  MoveL 4606 to (37.53, 58.52, -241.21) mm, rotated rx 42.04 ry 15.1 rz -114.75 deg; joints [-18.121, -37.551, 103.007, 143.689, 51.93, -28.848, -355]
  MoveL 4607 to (37.12, 58.35, -241.17) mm, rotated rx 42.04 ry 15.1 rz -114.75 deg; joints [-18.122, -37.581, 103.033, 143.686, 51.926, -28.844, -355]
  MoveL 4608 to (36.72, 58.21, -241.12) mm, rotated rx 42.04 ry 15.1 rz -114.75 deg; joints [-18.121, -37.609, 103.056, 143.684, 51.922, -28.841, -355]
  MoveL 4609 to (36.33, 58.09, -241.05) mm, rotated rx 42.04 ry 15.1 rz -114.75 deg; joints [-18.12, -37.637, 103.078, 143.683, 51.917, -28.837, -355]
  MoveL 4610 to (35.92, 57.93, -241) mm, rotated rx 42.04 ry 15.1 rz -114.75 deg; joints [-18.12, -37.667, 103.103, 143.681, 51.913, -28.833, -355]
  MoveL 4611 to (35.45, 57.73, -240.98) mm, rotated rx 42.04 ry 15.1 rz -114.75 deg; joints [-18.121, -37.701, 103.132, 143.677, 51.91, -28.829, -355]
  MoveL 4612 to (30.23, 55.38, -240.97) mm, rotated rx 42.04 ry 15.1 rz -114.75 deg; joints [-18.146, -38.084, 103.466, 143.625, 51.876, -28.782, -355]
  MoveL 4613 to (29.53, 55.08, -240.96) mm, rotated rx 42.04 ry 15.1 rz -114.75 deg; joints [-18.149, -38.136, 103.51, 143.618, 51.871, -28.775, -355]
  MoveL 4614 to (28.91, 54.84, -240.95) mm, rotated rx 42.04 ry 15.1 rz -114.75 deg; joints [-18.151, -38.179, 103.545, 143.612, 51.865, -28.767, -355]
  MoveL 4615 to (28.35, 54.72, -240.94) mm, rotated rx 42.04 ry 15.1 rz -114.75 deg; joints [-18.152, -38.217, 103.57, 143.604, 51.854, -28.757, -355]
  MoveL 4616 to (27.81, 54.68, -240.9) mm, rotated rx 42.04 ry 15.1 rz -114.75 deg; joints [-18.151, -38.251, 103.587, 143.598, 51.841, -28.745, -355]
  MoveL 4617 to (27.48, 54.71, -240.74) mm, rotated rx 42.04 ry 15.1 rz -114.75 deg; joints [-18.145, -38.271, 103.595, 143.599, 51.83, -28.739, -355]
  MoveL 4618 to (27.48, 54.74, -240.43) mm, rotated rx 42.04 ry 15.1 rz -114.75 deg; joints [-18.133, -38.272, 103.6, 143.614, 51.829, -28.746, -355]
  MoveL 4619 to (27.85, 54.75, -239.94) mm, rotated rx 42.04 ry 15.1 rz -114.75 deg; joints [-18.115, -38.254, 103.6, 143.645, 51.84, -28.768, -355]
  MoveL 4620 to (27.62, 55.34, -238.97) mm, rotated rx 42.04 ry 15.1 rz -114.75 deg; joints [-18.073, -38.258, 103.576, 143.68, 51.806, -28.764, -355]
  MoveL 4621 to (25.78, 55.69, -238.67) mm, rotated rx 42.04 ry 15.1 rz -114.75 deg; joints [-18.06, -38.36, 103.595, 143.657, 51.737, -28.707, -355]
  MoveL 4622 to (23.85, 56.05, -238.46) mm, rotated rx 42.04 ry 15.1 rz -114.75 deg; joints [-18.051, -38.466, 103.614, 143.627, 51.664, -28.646, -355]
  MoveL 4623 to (21.76, 56.41, -238.34) mm, rotated rx 42.04 ry 15.1 rz -114.75 deg; joints [-18.044, -38.581, 103.633, 143.59, 51.586, -28.576, -355]
  MoveL 4624 to (17.55, 57.12, -238.34) mm, rotated rx 42.04 ry 15.1 rz -114.75 deg; joints [-18.041, -38.81, 103.669, 143.503, 51.43, -28.431, -355]
  MoveL 4625 to (15.59, 57.45, -238.25) mm, rotated rx 42.04 ry 15.1 rz -114.75 deg; joints [-18.036, -38.916, 103.687, 143.466, 51.357, -28.366, -355]
  MoveL 4626 to (13.49, 57.8, -238.25) mm, rotated rx 42.04 ry 15.1 rz -114.75 deg; joints [-18.034, -39.031, 103.704, 143.422, 51.279, -28.292, -355]
  MoveL 4627 to (11.38, 58.25, -238.25) mm, rotated rx 42.04 ry 15.1 rz -114.75 deg; joints [-18.032, -39.142, 103.712, 143.376, 51.195, -28.215, -355]
  MoveL 4628 to (8.9, 58.83, -238.07) mm, rotated rx 42.04 ry 15.1 rz -114.75 deg; joints [-18.022, -39.273, 103.721, 143.329, 51.095, -28.126, -355]
  MoveL 4629 to (6.68, 59.07, -237.84) mm, rotated rx 42.04 ry 15.1 rz -114.75 deg; joints [-18.013, -39.398, 103.755, 143.295, 51.019, -28.059, -355]
  MoveL 4630 to (4.53, 59.33, -237.72) mm, rotated rx 42.04 ry 15.1 rz -114.75 deg; joints [-18.007, -39.519, 103.782, 143.257, 50.942, -27.99, -355]
  MoveL 4631 to (2.42, 59.68, -237.61) mm, rotated rx 42.04 ry 15.1 rz -114.75 deg; joints [-18.002, -39.633, 103.799, 143.216, 50.863, -27.918, -355]
  MoveL 4632 to (0.32, 60.02, -237.4) mm, rotated rx 42.04 ry 15.1 rz -114.75 deg; joints [-17.992, -39.748, 103.819, 143.181, 50.785, -27.848, -355]
  MoveL 4633 to (-1.79, 60.37, -237.29) mm, rotated rx 42.04 ry 15.1 rz -114.75 deg; joints [-17.986, -39.863, 103.837, 143.14, 50.705, -27.776, -355]
  MoveL 4634 to (-3.89, 60.71, -237.18) mm, rotated rx 42.04 ry 15.1 rz -114.75 deg; joints [-17.981, -39.977, 103.854, 143.099, 50.626, -27.703, -355]
  MoveL 4635 to (-6, 61.04, -236.97) mm, rotated rx 42.04 ry 15.1 rz -114.75 deg; joints [-17.971, -40.092, 103.874, 143.063, 50.548, -27.633, -355]
  MoveL 4636 to (-8.11, 61.38, -236.86) mm, rotated rx 42.04 ry 15.1 rz -114.75 deg; joints [-17.966, -40.206, 103.891, 143.022, 50.468, -27.56, -355]
  MoveL 4637 to (-10.21, 61.72, -236.76) mm, rotated rx 42.04 ry 15.1 rz -114.75 deg; joints [-17.96, -40.32, 103.907, 142.98, 50.389, -27.486, -355]
  MoveL 4638 to (-12.32, 62.04, -236.55) mm, rotated rx 42.04 ry 15.1 rz -114.75 deg; joints [-17.951, -40.436, 103.928, 142.943, 50.311, -27.416, -355]
  MoveL 4639 to (-14.43, 62.37, -236.45) mm, rotated rx 42.04 ry 15.1 rz -114.75 deg; joints [-17.946, -40.55, 103.944, 142.9, 50.231, -27.342, -355]
  MoveL 4640 to (-16.27, 62.58, -236.19) mm, rotated rx 42.04 ry 15.1 rz -114.75 deg; joints [-17.936, -40.653, 103.968, 142.873, 50.165, -27.284, -355]
  MoveL 4641 to (-17.93, 62.72, -235.82) mm, rotated rx 42.04 ry 15.1 rz -114.75 deg; joints [-17.922, -40.749, 103.997, 142.855, 50.108, -27.238, -355]
  MoveL 4642 to (-19.46, 62.77, -235.32) mm, rotated rx 42.04 ry 15.1 rz -114.75 deg; joints [-17.904, -40.841, 104.034, 142.849, 50.06, -27.203, -355]
  MoveL 4643 to (-18.41, 62.34, -234.48) mm, rotated rx 42.04 ry 15.1 rz -114.75 deg; joints [-17.875, -40.801, 104.069, 142.921, 50.112, -27.276, -355]
  MoveL 4644 to (-18.73, 62.4, -234.45) mm, rotated rx 42.04 ry 15.1 rz -114.75 deg; joints [-17.874, -40.819, 104.071, 142.915, 50.099, -27.264, -355]
  MoveL 4645 to (-19.05, 62.49, -234.41) mm, rotated rx 42.04 ry 15.1 rz -114.75 deg; joints [-17.872, -40.835, 104.071, 142.909, 50.085, -27.252, -355]
  MoveL 4646 to (-19.37, 62.66, -234.35) mm, rotated rx 42.04 ry 15.1 rz -114.75 deg; joints [-17.869, -40.848, 104.063, 142.902, 50.067, -27.237, -355]
  MoveL 4647 to (-19.71, 62.9, -234.31) mm, rotated rx 42.04 ry 15.1 rz -114.75 deg; joints [-17.865, -40.861, 104.05, 142.893, 50.046, -27.218, -355]
  MoveL 4648 to (-20.08, 63.21, -234.29) mm, rotated rx 42.04 ry 15.1 rz -114.75 deg; joints [-17.862, -40.873, 104.03, 142.881, 50.02, -27.195, -355]
  MoveL 4649 to (-23.51, 66.44, -234.29) mm, rotated rx 42.04 ry 15.1 rz -114.75 deg; joints [-17.836, -40.967, 103.812, 142.753, 49.763, -26.96, -355]
  MoveL 4650 to (-23.82, 66.7, -234.26) mm, rotated rx 42.04 ry 15.1 rz -114.75 deg; joints [-17.833, -40.977, 103.796, 142.744, 49.742, -26.941, -355]
  MoveL 4651 to (-24.2, 67.06, -234.26) mm, rotated rx 42.04 ry 15.1 rz -114.75 deg; joints [-17.83, -40.987, 103.771, 142.729, 49.714, -26.915, -355]
  MoveL 4652 to (-24.97, 67.75, -234.22) mm, rotated rx 42.04 ry 15.1 rz -114.75 deg; joints [-17.823, -41.01, 103.726, 142.703, 49.658, -26.865, -355]
  MoveL 4653 to (-26.87, 69.55, -234.22) mm, rotated rx 42.04 ry 15.1 rz -114.75 deg; joints [-17.808, -41.061, 103.604, 142.631, 49.516, -26.733, -355]
  MoveL 4654 to (-27.66, 70.21, -234.21) mm, rotated rx 42.04 ry 15.1 rz -114.75 deg; joints [-17.802, -41.085, 103.56, 142.603, 49.461, -26.682, -355]
  MoveL 4655 to (-28.72, 71.19, -234.27) mm, rotated rx 42.04 ry 15.1 rz -114.75 deg; joints [-17.797, -41.114, 103.493, 142.559, 49.382, -26.608, -355]
  MoveL 4656 to (-29.48, 72.08, -234.53) mm, rotated rx 42.04 ry 15.1 rz -114.75 deg; joints [-17.799, -41.126, 103.422, 142.513, 49.318, -26.541, -355]
  MoveL 4657 to (-29.94, 72.89, -234.97) mm, rotated rx 42.04 ry 15.1 rz -114.75 deg; joints [-17.809, -41.121, 103.35, 142.466, 49.266, -26.481, -355]
  MoveL 4658 to (-30.05, 73.26, -235.26) mm, rotated rx 42.04 ry 15.1 rz -114.75 deg; joints [-17.816, -41.112, 103.312, 142.442, 49.246, -26.455, -355]
  MoveL 4659 to (-30.09, 73.62, -235.59) mm, rotated rx 42.04 ry 15.1 rz -114.75 deg; joints [-17.826, -41.1, 103.275, 142.417, 49.228, -26.43, -355]
  MoveL 4660 to (-29.94, 74.26, -236.4) mm, rotated rx 42.04 ry 15.1 rz -114.75 deg; joints [-17.85, -41.062, 103.197, 142.367, 49.204, -26.386, -355]
  MoveL 4661 to (-29.48, 74.81, -237.4) mm, rotated rx 42.04 ry 15.1 rz -114.75 deg; joints [-17.882, -41.008, 103.117, 142.315, 49.193, -26.349, -355]
  MoveL 4662 to (-27.66, 75.67, -239.96) mm, rotated rx 42.04 ry 15.1 rz -114.75 deg; joints [-17.968, -40.851, 102.951, 142.207, 49.21, -26.3, -355]
  MoveL 4663 to (-25.28, 75.96, -242.53) mm, rotated rx 42.04 ry 15.1 rz -114.75 deg; joints [-18.059, -40.68, 102.822, 142.12, 49.269, -26.29, -355]
  MoveL 4664 to (-23, 75.48, -244.36) mm, rotated rx 42.04 ry 15.1 rz -114.75 deg; joints [-18.129, -40.547, 102.78, 142.084, 49.361, -26.329, -355]
  MoveL 4665 to (-21.89, 74.94, -245) mm, rotated rx 42.04 ry 15.1 rz -114.75 deg; joints [-18.157, -40.495, 102.792, 142.084, 49.42, -26.368, -355]
  MoveL 4666 to (-20.81, 74.21, -245.46) mm, rotated rx 42.04 ry 15.1 rz -114.75 deg; joints [-18.18, -40.453, 102.826, 142.097, 49.486, -26.418, -355]
  MoveL 4667 to (-18.73, 72.17, -245.82) mm, rotated rx 42.04 ry 15.1 rz -114.75 deg; joints [-18.21, -40.396, 102.958, 142.159, 49.644, -26.556, -355]
  MoveL 4668 to (-16.71, 69.76, -245.82) mm, rotated rx 42.04 ry 15.1 rz -114.75 deg; joints [-18.23, -40.358, 103.132, 142.245, 49.817, -26.717, -355]
  MoveL 4669 to (-16.04, 68.99, -245.84) mm, rotated rx 42.04 ry 15.1 rz -114.75 deg; joints [-18.237, -40.344, 103.186, 142.272, 49.873, -26.768, -355]
  MoveL 4670 to (-15.37, 68.19, -245.84) mm, rotated rx 42.04 ry 15.1 rz -114.75 deg; joints [-18.244, -40.331, 103.244, 142.3, 49.93, -26.821, -355]
  MoveL 4671 to (-15.04, 67.81, -245.84) mm, rotated rx 42.04 ry 15.1 rz -114.75 deg; joints [-18.247, -40.325, 103.271, 142.313, 49.958, -26.846, -355]
  MoveL 4672 to (-14.61, 67.31, -245.87) mm, rotated rx 42.04 ry 15.1 rz -114.75 deg; joints [-18.253, -40.316, 103.306, 142.33, 49.994, -26.879, -355]
  MoveL 4673 to (-14.2, 66.87, -245.93) mm, rotated rx 42.04 ry 15.1 rz -114.75 deg; joints [-18.258, -40.306, 103.335, 142.343, 50.027, -26.908, -355]
  MoveL 4674 to (-13.85, 66.51, -246) mm, rotated rx 42.04 ry 15.1 rz -114.75 deg; joints [-18.264, -40.296, 103.358, 142.353, 50.054, -26.931, -355]
  MoveL 4675 to (-13.52, 66.18, -246.05) mm, rotated rx 42.04 ry 15.1 rz -114.75 deg; joints [-18.269, -40.287, 103.38, 142.363, 50.08, -26.953, -355]
  MoveL 4676 to (-13.21, 65.84, -246.08) mm, rotated rx 42.04 ry 15.1 rz -114.75 deg; joints [-18.273, -40.28, 103.403, 142.373, 50.105, -26.975, -355]
  MoveL 4677 to (-12.2, 64.63, -246.08) mm, rotated rx 42.04 ry 15.1 rz -114.75 deg; joints [-18.283, -40.26, 103.489, 142.415, 50.192, -27.055, -355]
  MoveL 4678 to (-11.86, 64.26, -246.1) mm, rotated rx 42.04 ry 15.1 rz -114.75 deg; joints [-18.287, -40.252, 103.514, 142.428, 50.219, -27.08, -355]
  MoveL 4679 to (-11.55, 63.95, -246.13) mm, rotated rx 42.04 ry 15.1 rz -114.75 deg; joints [-18.29, -40.244, 103.535, 142.438, 50.243, -27.101, -355]
  MoveL 4680 to (-11.26, 63.7, -246.17) mm, rotated rx 42.04 ry 15.1 rz -114.75 deg; joints [-18.294, -40.234, 103.55, 142.446, 50.264, -27.118, -355]
  MoveL 4681 to (-10.99, 63.56, -246.24) mm, rotated rx 42.04 ry 15.1 rz -114.75 deg; joints [-18.298, -40.222, 103.555, 142.451, 50.278, -27.13, -355]
  MoveL 4682 to (-10.73, 63.46, -246.31) mm, rotated rx 42.04 ry 15.1 rz -114.75 deg; joints [-18.301, -40.21, 103.557, 142.454, 50.29, -27.14, -355]
  MoveL 4683 to (-11.92, 64.52, -247.11) mm, rotated rx 42.04 ry 15.1 rz -114.75 deg; joints [-18.322, -40.238, 103.47, 142.371, 50.205, -27.039, -355]
  MoveL 4684 to (-10.23, 63.99, -247.52) mm, rotated rx 42.04 ry 15.1 rz -114.75 deg; joints [-18.341, -40.153, 103.473, 142.393, 50.28, -27.101, -355]
  MoveL 4685 to (-8.44, 63.45, -247.78) mm, rotated rx 42.04 ry 15.1 rz -114.75 deg; joints [-18.354, -40.062, 103.477, 142.425, 50.359, -27.17, -355]
  MoveL 4686 to (-6.51, 62.9, -247.96) mm, rotated rx 42.04 ry 15.1 rz -114.75 deg; joints [-18.364, -39.965, 103.481, 142.464, 50.442, -27.245, -355]
  MoveL 4687 to (-4.46, 62.34, -248.16) mm, rotated rx 42.04 ry 15.1 rz -114.75 deg; joints [-18.375, -39.861, 103.483, 142.504, 50.529, -27.324, -355]
  MoveL 4688 to (-2.4, 61.76, -248.25) mm, rotated rx 42.04 ry 15.1 rz -114.75 deg; joints [-18.383, -39.758, 103.489, 142.55, 50.617, -27.406, -355]
  MoveL 4689 to (-0.35, 61.17, -248.35) mm, rotated rx 42.04 ry 15.1 rz -114.75 deg; joints [-18.39, -39.655, 103.494, 142.595, 50.705, -27.488, -355]
  MoveL 4690 to (1.71, 60.6, -248.55) mm, rotated rx 42.04 ry 15.1 rz -114.75 deg; joints [-18.401, -39.55, 103.496, 142.635, 50.793, -27.566, -355]
  MoveL 4691 to (3.76, 60.01, -248.65) mm, rotated rx 42.04 ry 15.1 rz -114.75 deg; joints [-18.409, -39.447, 103.501, 142.679, 50.881, -27.647, -355]
  MoveL 4692 to (5.81, 59.42, -248.75) mm, rotated rx 42.04 ry 15.1 rz -114.75 deg; joints [-18.416, -39.343, 103.505, 142.723, 50.969, -27.728, -355]
  MoveL 4693 to (7.86, 58.83, -248.95) mm, rotated rx 42.04 ry 15.1 rz -114.75 deg; joints [-18.428, -39.239, 103.507, 142.762, 51.056, -27.806, -355]
  MoveL 4694 to (11.96, 57.64, -249.15) mm, rotated rx 42.04 ry 15.1 rz -114.75 deg; joints [-18.443, -39.032, 103.515, 142.849, 51.232, -27.966, -355]
  MoveL 4695 to (13.68, 57.13, -249.36) mm, rotated rx 42.04 ry 15.1 rz -114.75 deg; joints [-18.454, -38.944, 103.516, 142.879, 51.306, -28.03, -355]
  MoveL 4696 to (15.57, 56.62, -249.43) mm, rotated rx 42.04 ry 15.1 rz -114.75 deg; joints [-18.46, -38.846, 103.516, 142.919, 51.385, -28.103, -355]
  MoveL 4697 to (17.57, 56.14, -249.44) mm, rotated rx 42.04 ry 15.1 rz -114.75 deg; joints [-18.464, -38.742, 103.512, 142.963, 51.466, -28.178, -355]
  MoveL 4698 to (20.13, 55.38, -249.55) mm, rotated rx 42.04 ry 15.1 rz -114.75 deg; joints [-18.473, -38.612, 103.517, 143.016, 51.576, -28.278, -355]
  MoveL 4699 to (22.57, 54.54, -249.64) mm, rotated rx 42.04 ry 15.1 rz -114.75 deg; joints [-18.482, -38.492, 103.532, 143.07, 51.686, -28.378, -355]
  MoveL 4700 to (24.68, 53.87, -249.74) mm, rotated rx 42.04 ry 15.1 rz -114.75 deg; joints [-18.49, -38.386, 103.538, 143.113, 51.778, -28.46, -355]
  MoveL 4701 to (26.64, 53.28, -249.91) mm, rotated rx 42.04 ry 15.1 rz -114.75 deg; joints [-18.501, -38.286, 103.54, 143.149, 51.862, -28.534, -355]
  MoveL 4702 to (28.45, 52.71, -250.19) mm, rotated rx 42.04 ry 15.1 rz -114.75 deg; joints [-18.515, -38.192, 103.54, 143.177, 51.941, -28.599, -355]
  MoveL 4703 to (30.26, 52.15, -250.48) mm, rotated rx 42.04 ry 15.1 rz -114.75 deg; joints [-18.53, -38.099, 103.54, 143.203, 52.019, -28.664, -355]
  MoveL 4704 to (32.04, 51.55, -250.77) mm, rotated rx 42.04 ry 15.1 rz -114.75 deg; joints [-18.545, -38.007, 103.543, 143.229, 52.098, -28.729, -355]
  MoveL 4705 to (33.94, 50.95, -250.93) mm, rotated rx 42.04 ry 15.1 rz -114.75 deg; joints [-18.555, -37.91, 103.545, 143.264, 52.18, -28.8, -355]
  MoveL 4706 to (34.26, 50.38, -251.55) mm, rotated rx 42.04 ry 15.1 rz -114.75 deg; joints [-18.583, -37.903, 103.573, 143.248, 52.216, -28.815, -355]
  MoveL 4707 to (33.95, 50.33, -251.86) mm, rotated rx 42.04 ry 15.1 rz -114.75 deg; joints [-18.595, -37.92, 103.579, 143.228, 52.209, -28.801, -355]
  MoveL 4708 to (33.93, 50.29, -252.05) mm, rotated rx 42.04 ry 15.1 rz -114.75 deg; joints [-18.603, -37.921, 103.579, 143.218, 52.21, -28.797, -355]
  MoveL 4709 to (34.18, 50.27, -252.15) mm, rotated rx 42.04 ry 15.1 rz -114.75 deg; joints [-18.607, -37.906, 103.572, 143.218, 52.218, -28.802, -355]
  MoveL 4710 to (34.62, 50.32, -252.17) mm, rotated rx 42.04 ry 15.1 rz -114.75 deg; joints [-18.606, -37.878, 103.556, 143.224, 52.228, -28.812, -355]
  MoveL 4711 to (35.1, 50.41, -252.17) mm, rotated rx 42.04 ry 15.1 rz -114.75 deg; joints [-18.605, -37.846, 103.536, 143.231, 52.237, -28.821, -355]
  MoveL 4712 to (36.04, 50.7, -252.2) mm, rotated rx 42.04 ry 15.1 rz -114.75 deg; joints [-18.603, -37.781, 103.487, 143.241, 52.249, -28.834, -355]
  MoveL 4713 to (37.53, 51.18, -252.2) mm, rotated rx 42.04 ry 15.1 rz -114.75 deg; joints [-18.598, -37.677, 103.409, 143.259, 52.269, -28.855, -355]
  MoveL 4714 to (38.48, 51.44, -252.22) mm, rotated rx 42.04 ry 15.1 rz -114.75 deg; joints [-18.595, -37.613, 103.362, 143.27, 52.282, -28.87, -355]
  MoveL 4715 to (39.48, 51.75, -252.22) mm, rotated rx 42.04 ry 15.1 rz -114.75 deg; joints [-18.591, -37.543, 103.31, 143.283, 52.295, -28.884, -355]
  MoveL 4716 to (39.97, 51.9, -252.23) mm, rotated rx 42.04 ry 15.1 rz -114.75 deg; joints [-18.59, -37.509, 103.284, 143.288, 52.301, -28.891, -355]
  MoveL 4717 to (40.42, 52.03, -252.26) mm, rotated rx 42.04 ry 15.1 rz -114.75 deg; joints [-18.59, -37.478, 103.261, 143.292, 52.308, -28.897, -355]
  MoveL 4718 to (40.85, 52.14, -252.31) mm, rotated rx 42.04 ry 15.1 rz -114.75 deg; joints [-18.59, -37.449, 103.24, 143.295, 52.314, -28.903, -355]
  MoveL 4719 to (41.24, 52.24, -252.37) mm, rotated rx 42.04 ry 15.1 rz -114.75 deg; joints [-18.591, -37.422, 103.22, 143.297, 52.32, -28.908, -355]
  MoveL 4720 to (41.65, 52.34, -252.43) mm, rotated rx 42.04 ry 15.1 rz -114.75 deg; joints [-18.592, -37.394, 103.2, 143.3, 52.327, -28.914, -355]
  MoveL 4721 to (42.09, 52.46, -252.46) mm, rotated rx 42.04 ry 15.1 rz -114.75 deg; joints [-18.592, -37.363, 103.177, 143.304, 52.333, -28.92, -355]
  MoveL 4722 to (42.55, 52.59, -252.48) mm, rotated rx 42.04 ry 15.1 rz -114.75 deg; joints [-18.591, -37.331, 103.154, 143.308, 52.339, -28.926, -355]
  MoveL 4723 to (42.98, 52.7, -252.53) mm, rotated rx 42.04 ry 15.1 rz -114.75 deg; joints [-18.591, -37.303, 103.133, 143.312, 52.346, -28.932, -355]
  MoveL 4724 to (43.37, 52.78, -252.59) mm, rotated rx 42.04 ry 15.1 rz -114.75 deg; joints [-18.593, -37.276, 103.115, 143.314, 52.353, -28.938, -355]
  MoveL 4725 to (43.77, 52.87, -252.64) mm, rotated rx 42.04 ry 15.1 rz -114.75 deg; joints [-18.593, -37.249, 103.095, 143.317, 52.359, -28.944, -355]
  MoveL 4726 to (44.2, 52.98, -252.67) mm, rotated rx 42.04 ry 15.1 rz -114.75 deg; joints [-18.593, -37.22, 103.074, 143.321, 52.366, -28.95, -355]
  MoveL 4727 to (44.7, 53.14, -252.67) mm, rotated rx 42.04 ry 15.1 rz -114.75 deg; joints [-18.591, -37.185, 103.048, 143.327, 52.372, -28.957, -355]
  MoveL 4728 to (47.54, 53.78, -253.03) mm, rotated rx 42.04 ry 15.1 rz -114.75 deg; joints [-18.597, -36.992, 102.912, 143.347, 52.419, -28.997, -355]
  MoveL 4729 to (48.83, 53.85, -253.47) mm, rotated rx 42.04 ry 15.1 rz -114.75 deg; joints [-18.611, -36.909, 102.862, 143.345, 52.449, -29.017, -355]
  MoveL 4730 to (50.03, 53.76, -254.09) mm, rotated rx 42.04 ry 15.1 rz -114.75 deg; joints [-18.634, -36.834, 102.825, 143.335, 52.485, -29.036, -355]
  MoveL 4731 to (52.15, 53.11, -255.87) mm, rotated rx 42.04 ry 15.1 rz -114.75 deg; joints [-18.705, -36.711, 102.788, 143.293, 52.571, -29.071, -355]
  MoveL 4732 to (53.9, 51.8, -258.37) mm, rotated rx 42.04 ry 15.1 rz -114.75 deg; joints [-18.809, -36.622, 102.8, 143.219, 52.677, -29.105, -355]
  MoveL 4733 to (54.89, 50.3, -260.86) mm, rotated rx 42.04 ry 15.1 rz -114.75 deg; joints [-18.915, -36.585, 102.849, 143.135, 52.772, -29.127, -355]
  MoveL 4734 to (54.95, 49.65, -261.84) mm, rotated rx 42.04 ry 15.1 rz -114.75 deg; joints [-18.957, -36.592, 102.882, 143.097, 52.803, -29.13, -355]
  MoveL 4735 to (54.71, 49.05, -262.64) mm, rotated rx 42.04 ry 15.1 rz -114.75 deg; joints [-18.993, -36.617, 102.922, 143.063, 52.823, -29.126, -355]
  MoveL 4736 to (54.48, 48.78, -262.98) mm, rotated rx 42.04 ry 15.1 rz -114.75 deg; joints [-19.008, -36.635, 102.944, 143.047, 52.83, -29.123, -355]
  MoveL 4737 to (54.18, 48.53, -263.27) mm, rotated rx 42.04 ry 15.1 rz -114.75 deg; joints [-19.021, -36.659, 102.967, 143.032, 52.833, -29.118, -355]
  MoveL 4738 to (53.36, 48.06, -263.71) mm, rotated rx 42.04 ry 15.1 rz -114.75 deg; joints [-19.043, -36.718, 103.019, 143.003, 52.832, -29.103, -355]
  MoveL 4739 to (52.24, 47.66, -263.98) mm, rotated rx 42.04 ry 15.1 rz -114.75 deg; joints [-19.058, -36.795, 103.077, 142.977, 52.821, -29.083, -355]
  MoveL 4740 to (50.83, 47.32, -264.07) mm, rotated rx 42.04 ry 15.1 rz -114.75 deg; joints [-19.065, -36.889, 103.14, 142.955, 52.799, -29.057, -355]
  MoveL 4741 to (48.26, 46.82, -264.07) mm, rotated rx 42.04 ry 15.1 rz -114.75 deg; joints [-19.072, -37.058, 103.25, 142.919, 52.753, -29.009, -355]
  MoveL 4742 to (47.82, 46.75, -264.04) mm, rotated rx 42.04 ry 15.1 rz -114.75 deg; joints [-19.072, -37.086, 103.268, 142.915, 52.744, -29.001, -355]
  MoveL 4743 to (47.42, 46.7, -263.99) mm, rotated rx 42.04 ry 15.1 rz -114.75 deg; joints [-19.071, -37.113, 103.284, 142.911, 52.736, -28.994, -355]
  MoveL 4744 to (47.04, 46.66, -263.92) mm, rotated rx 42.04 ry 15.1 rz -114.75 deg; joints [-19.069, -37.138, 103.299, 142.909, 52.727, -28.987, -355]
  MoveL 4745 to (46.61, 46.6, -263.87) mm, rotated rx 42.04 ry 15.1 rz -114.75 deg; joints [-19.068, -37.165, 103.316, 142.905, 52.719, -28.979, -355]
  MoveL 4746 to (46.12, 46.52, -263.83) mm, rotated rx 42.04 ry 15.1 rz -114.75 deg; joints [-19.068, -37.198, 103.336, 142.9, 52.709, -28.97, -355]
  MoveL 4747 to (45.6, 46.45, -263.77) mm, rotated rx 42.04 ry 15.1 rz -114.75 deg; joints [-19.067, -37.231, 103.357, 142.895, 52.698, -28.961, -355]
  MoveL 4748 to (45.06, 46.36, -263.76) mm, rotated rx 42.04 ry 15.1 rz -114.75 deg; joints [-19.067, -37.266, 103.379, 142.888, 52.688, -28.951, -355]
  MoveL 4749 to (44.43, 46.23, -263.77) mm, rotated rx 42.04 ry 15.1 rz -114.75 deg; joints [-19.07, -37.308, 103.406, 142.879, 52.677, -28.938, -355]
  MoveL 4750 to (43.59, 46.04, -263.84) mm, rotated rx 42.04 ry 15.1 rz -114.75 deg; joints [-19.075, -37.364, 103.442, 142.864, 52.663, -28.922, -355]
  MoveL 4751 to (43.07, 45.94, -263.84) mm, rotated rx 42.04 ry 15.1 rz -114.75 deg; joints [-19.076, -37.398, 103.464, 142.857, 52.653, -28.912, -355]
  MoveL 4752 to (42.58, 45.85, -263.83) mm, rotated rx 42.04 ry 15.1 rz -114.75 deg; joints [-19.077, -37.43, 103.484, 142.85, 52.644, -28.903, -355]
  MoveL 4753 to (42.12, 45.77, -263.81) mm, rotated rx 42.04 ry 15.1 rz -114.75 deg; joints [-19.077, -37.46, 103.503, 142.845, 52.635, -28.894, -355]
  MoveL 4754 to (41.71, 45.71, -263.76) mm, rotated rx 42.04 ry 15.1 rz -114.75 deg; joints [-19.076, -37.487, 103.52, 142.841, 52.626, -28.886, -355]
  MoveL 4755 to (41.31, 45.68, -263.7) mm, rotated rx 42.04 ry 15.1 rz -114.75 deg; joints [-19.075, -37.512, 103.534, 142.838, 52.617, -28.878, -355]
  MoveL 4756 to (40.89, 45.69, -263.65) mm, rotated rx 42.04 ry 15.1 rz -114.75 deg; joints [-19.073, -37.538, 103.545, 142.833, 52.605, -28.868, -355]
  MoveL 4757 to (40.48, 45.74, -263.59) mm, rotated rx 42.04 ry 15.1 rz -114.75 deg; joints [-19.071, -37.561, 103.552, 142.828, 52.591, -28.856, -355]
  MoveL 4758 to (40.27, 45.83, -263.43) mm, rotated rx 42.04 ry 15.1 rz -114.75 deg; joints [-19.064, -37.573, 103.553, 142.831, 52.582, -28.851, -355]
  MoveL 4759 to (40.37, 45.89, -263.12) mm, rotated rx 42.04 ry 15.1 rz -114.75 deg; joints [-19.052, -37.568, 103.553, 142.847, 52.582, -28.86, -355]
  MoveL 4760 to (40.81, 45.91, -262.62) mm, rotated rx 42.04 ry 15.1 rz -114.75 deg; joints [-19.033, -37.546, 103.552, 142.879, 52.595, -28.884, -355]
  MoveL 4761 to (39.98, 46.22, -261.77) mm, rotated rx 42.04 ry 15.1 rz -114.75 deg; joints [-18.999, -37.594, 103.565, 142.902, 52.558, -28.871, -355]
  MoveL 4762 to (36.04, 47.87, -261.77) mm, rotated rx 42.04 ry 15.1 rz -114.75 deg; joints [-18.986, -37.781, 103.518, 142.809, 52.369, -28.698, -355]
  MoveL 4763 to (34.2, 48.65, -261.71) mm, rotated rx 42.04 ry 15.1 rz -114.75 deg; joints [-18.978, -37.869, 103.497, 142.768, 52.28, -28.618, -355]
  MoveL 4764 to (32.37, 49.43, -261.56) mm, rotated rx 42.04 ry 15.1 rz -114.75 deg; joints [-18.966, -37.956, 103.476, 142.73, 52.191, -28.54, -355]
  MoveL 4765 to (30.26, 50.34, -261.36) mm, rotated rx 42.04 ry 15.1 rz -114.75 deg; joints [-18.952, -38.057, 103.452, 142.689, 52.088, -28.451, -355]
  MoveL 4766 to (28.27, 51.2, -261.15) mm, rotated rx 42.04 ry 15.1 rz -114.75 deg; joints [-18.937, -38.152, 103.43, 142.65, 51.991, -28.367, -355]
  MoveL 4767 to (26.26, 52.05, -261.05) mm, rotated rx 42.04 ry 15.1 rz -114.75 deg; joints [-18.927, -38.247, 103.406, 142.605, 51.894, -28.279, -355]
  MoveL 4768 to (24.29, 52.87, -261.05) mm, rotated rx 42.04 ry 15.1 rz -114.75 deg; joints [-18.921, -38.339, 103.38, 142.557, 51.799, -28.191, -355]
  MoveL 4769 to (22.46, 53.64, -260.98) mm, rotated rx 42.04 ry 15.1 rz -114.75 deg; joints [-18.912, -38.425, 103.358, 142.514, 51.71, -28.11, -355]
  MoveL 4770 to (20.73, 54.36, -260.86) mm, rotated rx 42.04 ry 15.1 rz -114.75 deg; joints [-18.903, -38.507, 103.338, 142.477, 51.627, -28.035, -355]
  MoveL 4771 to (18.84, 55.15, -260.8) mm, rotated rx 42.04 ry 15.1 rz -114.75 deg; joints [-18.894, -38.596, 103.314, 142.432, 51.536, -27.952, -355]
  MoveL 4772 to (16.87, 55.97, -260.62) mm, rotated rx 42.04 ry 15.1 rz -114.75 deg; joints [-18.881, -38.689, 103.291, 142.391, 51.441, -27.867, -355]
  MoveL 4773 to (12.93, 57.61, -260.44) mm, rotated rx 42.04 ry 15.1 rz -114.75 deg; joints [-18.862, -38.873, 103.241, 142.299, 51.25, -27.692, -355]
  MoveL 4774 to (10.96, 58.43, -260.26) mm, rotated rx 42.04 ry 15.1 rz -114.75 deg; joints [-18.849, -38.966, 103.218, 142.258, 51.155, -27.607, -355]
  MoveL 4775 to (8.98, 59.24, -260.08) mm, rotated rx 42.04 ry 15.1 rz -114.75 deg; joints [-18.836, -39.059, 103.195, 142.215, 51.06, -27.521, -355]
  MoveL 4776 to (7.02, 60.06, -260.08) mm, rotated rx 42.04 ry 15.1 rz -114.75 deg; joints [-18.83, -39.149, 103.166, 142.164, 50.964, -27.43, -355]
  MoveL 4777 to (5.04, 60.87, -259.9) mm, rotated rx 42.04 ry 15.1 rz -114.75 deg; joints [-18.817, -39.242, 103.143, 142.121, 50.869, -27.344, -355]
  MoveL 4778 to (3.06, 61.67, -259.72) mm, rotated rx 42.04 ry 15.1 rz -114.75 deg; joints [-18.805, -39.334, 103.12, 142.077, 50.774, -27.258, -355]
  MoveL 4779 to (1.09, 62.49, -259.72) mm, rotated rx 42.04 ry 15.1 rz -114.75 deg; joints [-18.799, -39.424, 103.09, 142.025, 50.679, -27.166, -355]
  MoveL 4780 to (-0.73, 63.18, -259.53) mm, rotated rx 42.04 ry 15.1 rz -114.75 deg; joints [-18.786, -39.511, 103.073, 141.987, 50.594, -27.089, -355]
  MoveL 4781 to (-2.36, 63.72, -259.21) mm, rotated rx 42.04 ry 15.1 rz -114.75 deg; joints [-18.771, -39.592, 103.068, 141.962, 50.521, -27.027, -355]
  MoveL 4782 to (-3.83, 64.12, -258.74) mm, rotated rx 42.04 ry 15.1 rz -114.75 deg; joints [-18.751, -39.67, 103.074, 141.949, 50.459, -26.979, -355]
  MoveL 4783 to (-3.04, 63.61, -257.98) mm, rotated rx 42.04 ry 15.1 rz -114.75 deg; joints [-18.727, -39.647, 103.121, 142.013, 50.507, -27.045, -355]
  MoveL 4784 to (-3.4, 63.81, -257.97) mm, rotated rx 42.04 ry 15.1 rz -114.75 deg; joints [-18.725, -39.662, 103.111, 142.002, 50.487, -27.026, -355]
  MoveC 4785 to (-5.59, 66.61, -257.97) mm, rotated rx 42.04 ry 15.1 rz -114.75 deg; joints [-18.701, -39.7, 102.909, 141.909, 50.292, -26.846, -355] to (-7.54, 69.58, -257.97) mm, rotated rx 42.04 ry 15.1 rz -114.75 deg; joints [-18.674, -39.717, 102.687, 141.817, 50.096, -26.665, -355]
  MoveL 4786 to (-7.54, 69.58, -257.97) mm, rotated rx 42.04 ry 15.1 rz -114.75 deg; joints [-18.674, -39.717, 102.687, 141.817, 50.096, -26.665, -355]
  MoveL 4787 to (-7.81, 69.96, -257.95) mm, rotated rx 42.04 ry 15.1 rz -114.75 deg; joints [-18.67, -39.721, 102.658, 141.805, 50.07, -26.642, -355]
  MoveL 4788 to (-8.07, 70.3, -257.9) mm, rotated rx 42.04 ry 15.1 rz -114.75 deg; joints [-18.665, -39.725, 102.635, 141.797, 50.047, -26.622, -355]
  MoveL 4789 to (-8.32, 70.62, -257.84) mm, rotated rx 42.04 ry 15.1 rz -114.75 deg; joints [-18.66, -39.73, 102.613, 141.789, 50.024, -26.602, -355]
  MoveL 4790 to (-8.58, 70.97, -257.79) mm, rotated rx 42.04 ry 15.1 rz -114.75 deg; joints [-18.656, -39.734, 102.589, 141.779, 50, -26.581, -355]
  MoveL 4791 to (-8.85, 71.35, -257.76) mm, rotated rx 42.04 ry 15.1 rz -114.75 deg; joints [-18.651, -39.738, 102.561, 141.768, 49.974, -26.558, -355]
  MoveL 4792 to (-9.15, 71.78, -257.75) mm, rotated rx 42.04 ry 15.1 rz -114.75 deg; joints [-18.647, -39.741, 102.529, 141.755, 49.946, -26.532, -355]
  MoveL 4793 to (-9.72, 72.66, -257.75) mm, rotated rx 42.04 ry 15.1 rz -114.75 deg; joints [-18.639, -39.746, 102.463, 141.728, 49.888, -26.478, -355]
  MoveL 4794 to (-10.48, 73.9, -257.84) mm, rotated rx 42.04 ry 15.1 rz -114.75 deg; joints [-18.632, -39.748, 102.366, 141.685, 49.808, -26.401, -355]
  MoveL 4795 to (-10.99, 74.99, -258.11) mm, rotated rx 42.04 ry 15.1 rz -114.75 deg; joints [-18.632, -39.739, 102.273, 141.64, 49.742, -26.332, -355]
  MoveL 4796 to (-11.26, 75.92, -258.57) mm, rotated rx 42.04 ry 15.1 rz -114.75 deg; joints [-18.641, -39.72, 102.185, 141.594, 49.691, -26.273, -355]
  MoveL 4797 to (-11.28, 76.69, -259.21) mm, rotated rx 42.04 ry 15.1 rz -114.75 deg; joints [-18.657, -39.69, 102.102, 141.546, 49.654, -26.222, -355]
  MoveL 4798 to (-11.07, 77.3, -260.03) mm, rotated rx 42.04 ry 15.1 rz -114.75 deg; joints [-18.681, -39.649, 102.024, 141.497, 49.632, -26.179, -355]
  MoveL 4799 to (-10.62, 77.75, -261.04) mm, rotated rx 42.04 ry 15.1 rz -114.75 deg; joints [-18.714, -39.598, 101.951, 141.447, 49.624, -26.146, -355]
  MoveL 4800 to (-8.98, 78.18, -263.6) mm, rotated rx 42.04 ry 15.1 rz -114.75 deg; joints [-18.803, -39.465, 101.82, 141.342, 49.651, -26.105, -355]
  MoveL 4801 to (-6.94, 77.93, -266.16) mm, rotated rx 42.04 ry 15.1 rz -114.75 deg; joints [-18.897, -39.331, 101.74, 141.258, 49.721, -26.105, -355]
  MoveL 4802 to (-5.99, 77.53, -267.16) mm, rotated rx 42.04 ry 15.1 rz -114.75 deg; joints [-18.937, -39.279, 101.733, 141.234, 49.767, -26.123, -355]
  MoveL 4803 to (-5.08, 76.94, -267.99) mm, rotated rx 42.04 ry 15.1 rz -114.75 deg; joints [-18.972, -39.237, 101.746, 141.222, 49.82, -26.152, -355]
  MoveL 4804 to (-4.2, 76.17, -268.63) mm, rotated rx 42.04 ry 15.1 rz -114.75 deg; joints [-19.002, -39.206, 101.782, 141.221, 49.881, -26.192, -355]
  MoveL 4805 to (-3.37, 75.22, -269.08) mm, rotated rx 42.04 ry 15.1 rz -114.75 deg; joints [-19.027, -39.184, 101.839, 141.233, 49.949, -26.245, -355]
  MoveL 4806 to (-1.84, 72.76, -269.45) mm, rotated rx 42.04 ry 15.1 rz -114.75 deg; joints [-19.062, -39.172, 102.016, 141.29, 50.108, -26.383, -355]
  MoveL 4807 to (-1.36, 71.83, -269.45) mm, rotated rx 42.04 ry 15.1 rz -114.75 deg; joints [-19.071, -39.174, 102.089, 141.317, 50.165, -26.437, -355]
  MoveL 4808 to (-1.12, 71.36, -269.46) mm, rotated rx 42.04 ry 15.1 rz -114.75 deg; joints [-19.075, -39.175, 102.125, 141.33, 50.194, -26.463, -355]
  MoveL 4809 to (-0.89, 70.95, -269.48) mm, rotated rx 42.04 ry 15.1 rz -114.75 deg; joints [-19.08, -39.175, 102.157, 141.341, 50.22, -26.487, -355]
  MoveL 4810 to (-0.67, 70.58, -269.53) mm, rotated rx 42.04 ry 15.1 rz -114.75 deg; joints [-19.085, -39.174, 102.183, 141.35, 50.243, -26.507, -355]
  MoveL 4811 to (-0.46, 70.24, -269.58) mm, rotated rx 42.04 ry 15.1 rz -114.75 deg; joints [-19.09, -39.172, 102.208, 141.357, 50.265, -26.526, -355]
  MoveL 4812 to (-0.24, 69.88, -269.63) mm, rotated rx 42.04 ry 15.1 rz -114.75 deg; joints [-19.095, -39.171, 102.234, 141.366, 50.288, -26.546, -355]
  MoveL 4813 to (-0.02, 69.47, -269.65) mm, rotated rx 42.04 ry 15.1 rz -114.75 deg; joints [-19.1, -39.171, 102.265, 141.376, 50.314, -26.57, -355]
  MoveL 4814 to (0.21, 69.03, -269.66) mm, rotated rx 42.04 ry 15.1 rz -114.75 deg; joints [-19.104, -39.172, 102.3, 141.389, 50.341, -26.595, -355]
  MoveL 4815 to (0.46, 68.53, -269.65) mm, rotated rx 42.04 ry 15.1 rz -114.75 deg; joints [-19.108, -39.173, 102.338, 141.403, 50.371, -26.623, -355]
  MoveL 4816 to (0.71, 68.06, -269.66) mm, rotated rx 42.04 ry 15.1 rz -114.75 deg; joints [-19.113, -39.174, 102.374, 141.416, 50.4, -26.65, -355]
  MoveL 4817 to (0.94, 67.63, -269.68) mm, rotated rx 42.04 ry 15.1 rz -114.75 deg; joints [-19.118, -39.174, 102.407, 141.427, 50.427, -26.674, -355]
  MoveL 4818 to (1.18, 67.22, -269.73) mm, rotated rx 42.04 ry 15.1 rz -114.75 deg; joints [-19.123, -39.173, 102.438, 141.437, 50.453, -26.697, -355]
  MoveL 4819 to (1.44, 66.79, -269.81) mm, rotated rx 42.04 ry 15.1 rz -114.75 deg; joints [-19.13, -39.171, 102.468, 141.446, 50.481, -26.72, -355]
  MoveL 4820 to (1.75, 66.27, -269.87) mm, rotated rx 42.04 ry 15.1 rz -114.75 deg; joints [-19.137, -39.168, 102.506, 141.458, 50.514, -26.749, -355]
  MoveL 4821 to (2.02, 65.77, -269.89) mm, rotated rx 42.04 ry 15.1 rz -114.75 deg; joints [-19.142, -39.168, 102.544, 141.471, 50.546, -26.778, -355]
  MoveL 4822 to (2.27, 65.3, -269.89) mm, rotated rx 42.04 ry 15.1 rz -114.75 deg; joints [-19.146, -39.169, 102.58, 141.484, 50.574, -26.804, -355]
  MoveL 4823 to (2.51, 64.83, -269.89) mm, rotated rx 42.04 ry 15.1 rz -114.75 deg; joints [-19.151, -39.17, 102.616, 141.497, 50.603, -26.831, -355]
  MoveL 4824 to (2.83, 64.26, -269.9) mm, rotated rx 42.04 ry 15.1 rz -114.75 deg; joints [-19.156, -39.17, 102.66, 141.513, 50.639, -26.864, -355]
  MoveL 4825 to (3.12, 63.75, -269.91) mm, rotated rx 42.04 ry 15.1 rz -114.75 deg; joints [-19.161, -39.168, 102.698, 141.527, 50.671, -26.893, -355]
  MoveL 4826 to (3.4, 63.33, -269.92) mm, rotated rx 42.04 ry 15.1 rz -114.75 deg; joints [-19.165, -39.165, 102.729, 141.54, 50.699, -26.919, -355]
  MoveL 4827 to (3.64, 63.08, -269.92) mm, rotated rx 42.04 ry 15.1 rz -114.75 deg; joints [-19.168, -39.159, 102.746, 141.549, 50.718, -26.936, -355]
  MoveL 4828 to (3.85, 62.92, -269.92) mm, rotated rx 42.04 ry 15.1 rz -114.75 deg; joints [-19.169, -39.152, 102.756, 141.556, 50.732, -26.949, -355]
  MoveL 4829 to (3.1, 63.48, -270.51) mm, rotated rx 42.04 ry 15.1 rz -114.75 deg; joints [-19.186, -39.172, 102.708, 141.501, 50.683, -26.887, -355]
  MoveL 4830 to (4.38, 63.09, -271.04) mm, rotated rx 42.04 ry 15.1 rz -114.75 deg; joints [-19.208, -39.105, 102.703, 141.506, 50.738, -26.927, -355]
  MoveL 4831 to (5.83, 62.49, -271.42) mm, rotated rx 42.04 ry 15.1 rz -114.75 deg; joints [-19.227, -39.035, 102.714, 141.526, 50.806, -26.984, -355]
  MoveL 4832 to (7.49, 61.69, -271.68) mm, rotated rx 42.04 ry 15.1 rz -114.75 deg; joints [-19.243, -38.961, 102.742, 141.559, 50.891, -27.059, -355]
  MoveL 4833 to (9.3, 60.72, -271.81) mm, rotated rx 42.04 ry 15.1 rz -114.75 deg; joints [-19.256, -38.883, 102.784, 141.604, 50.988, -27.149, -355]
  MoveL 4834 to (11.15, 59.72, -271.9) mm, rotated rx 42.04 ry 15.1 rz -114.75 deg; joints [-19.267, -38.805, 102.83, 141.652, 51.088, -27.242, -355]
  MoveL 4835 to (14.89, 57.67, -272.08) mm, rotated rx 42.04 ry 15.1 rz -114.75 deg; joints [-19.291, -38.647, 102.921, 141.749, 51.29, -27.43, -355]
  MoveL 4836 to (16.76, 56.65, -272.26) mm, rotated rx 42.04 ry 15.1 rz -114.75 deg; joints [-19.306, -38.566, 102.963, 141.793, 51.391, -27.521, -355]
  MoveL 4837 to (20.5, 54.59, -272.44) mm, rotated rx 42.04 ry 15.1 rz -114.75 deg; joints [-19.329, -38.406, 103.053, 141.887, 51.593, -27.708, -355]
  MoveL 4838 to (22.37, 53.57, -272.62) mm, rotated rx 42.04 ry 15.1 rz -114.75 deg; joints [-19.345, -38.325, 103.095, 141.93, 51.694, -27.798, -355]
  MoveL 4839 to (24.24, 52.53, -272.71) mm, rotated rx 42.04 ry 15.1 rz -114.75 deg; joints [-19.356, -38.245, 103.14, 141.976, 51.796, -27.891, -355]
  MoveL 4840 to (25.95, 51.56, -272.92) mm, rotated rx 42.04 ry 15.1 rz -114.75 deg; joints [-19.372, -38.171, 103.18, 142.013, 51.89, -27.974, -355]
  MoveL 4841 to (28.02, 50.42, -273.07) mm, rotated rx 42.04 ry 15.1 rz -114.75 deg; joints [-19.387, -38.081, 103.227, 142.061, 52.001, -28.074, -355]
  MoveL 4842 to (30.26, 49.18, -273.19) mm, rotated rx 42.04 ry 15.1 rz -114.75 deg; joints [-19.402, -37.984, 103.278, 142.116, 52.123, -28.184, -355]
  MoveL 4843 to (32.13, 48.14, -273.19) mm, rotated rx 42.04 ry 15.1 rz -114.75 deg; joints [-19.411, -37.903, 103.323, 142.165, 52.224, -28.278, -355]
  MoveL 4844 to (33.91, 47.15, -273.26) mm, rotated rx 42.04 ry 15.1 rz -114.75 deg; joints [-19.422, -37.826, 103.365, 142.209, 52.321, -28.366, -355]
  MoveL 4845 to (35.49, 46.25, -273.44) mm, rotated rx 42.04 ry 15.1 rz -114.75 deg; joints [-19.436, -37.756, 103.401, 142.242, 52.408, -28.442, -355]
  MoveL 4846 to (37.11, 45.31, -273.65) mm, rotated rx 42.04 ry 15.1 rz -114.75 deg; joints [-19.452, -37.686, 103.438, 142.275, 52.497, -28.519, -355]
  MoveL 4847 to (39.17, 44.15, -273.78) mm, rotated rx 42.04 ry 15.1 rz -114.75 deg; joints [-19.466, -37.595, 103.484, 142.322, 52.609, -28.618, -355]
  MoveL 4848 to (41.42, 42.9, -273.89) mm, rotated rx 42.04 ry 15.1 rz -114.75 deg; joints [-19.481, -37.496, 103.535, 142.375, 52.732, -28.727, -355]
  MoveL 4849 to (45.15, 40.83, -273.89) mm, rotated rx 42.04 ry 15.1 rz -114.75 deg; joints [-19.498, -37.332, 103.62, 142.47, 52.934, -28.911, -355]
  MoveL 4850 to (45.23, 40.52, -274.59) mm, rotated rx 42.04 ry 15.1 rz -114.75 deg; joints [-19.527, -37.33, 103.629, 142.442, 52.949, -28.908, -355]
  MoveL 4851 to (44.91, 40.55, -274.93) mm, rotated rx 42.04 ry 15.1 rz -114.75 deg; joints [-19.54, -37.345, 103.626, 142.419, 52.938, -28.889, -355]
  MoveL 4852 to (44.9, 40.54, -275.15) mm, rotated rx 42.04 ry 15.1 rz -114.75 deg; joints [-19.548, -37.344, 103.622, 142.408, 52.938, -28.883, -355]
  MoveL 4853 to (45.17, 40.49, -275.26) mm, rotated rx 42.04 ry 15.1 rz -114.75 deg; joints [-19.552, -37.328, 103.617, 142.407, 52.947, -28.889, -355]
  MoveL 4854 to (45.62, 40.47, -275.29) mm, rotated rx 42.04 ry 15.1 rz -114.75 deg; joints [-19.553, -37.301, 103.607, 142.414, 52.96, -28.902, -355]
  MoveL 4855 to (46.09, 40.48, -275.32) mm, rotated rx 42.04 ry 15.1 rz -114.75 deg; joints [-19.554, -37.272, 103.593, 142.421, 52.973, -28.914, -355]
  MoveL 4856 to (46.53, 40.49, -275.36) mm, rotated rx 42.04 ry 15.1 rz -114.75 deg; joints [-19.555, -37.245, 103.58, 142.425, 52.984, -28.924, -355]
  MoveL 4857 to (46.93, 40.49, -275.43) mm, rotated rx 42.04 ry 15.1 rz -114.75 deg; joints [-19.557, -37.221, 103.568, 142.429, 52.995, -28.933, -355]
  MoveL 4858 to (47.34, 40.5, -275.49) mm, rotated rx 42.04 ry 15.1 rz -114.75 deg; joints [-19.559, -37.195, 103.556, 142.433, 53.006, -28.942, -355]
  MoveL 4859 to (47.78, 40.52, -275.53) mm, rotated rx 42.04 ry 15.1 rz -114.75 deg; joints [-19.56, -37.167, 103.542, 142.438, 53.017, -28.952, -355]
  MoveL 4860 to (48.3, 40.55, -275.55) mm, rotated rx 42.04 ry 15.1 rz -114.75 deg; joints [-19.56, -37.135, 103.525, 142.445, 53.029, -28.964, -355]
  MoveL 4861 to (48.83, 40.56, -275.62) mm, rotated rx 42.04 ry 15.1 rz -114.75 deg; joints [-19.562, -37.102, 103.509, 142.451, 53.043, -28.976, -355]
  MoveL 4862 to (49.36, 40.59, -275.65) mm, rotated rx 42.04 ry 15.1 rz -114.75 deg; joints [-19.563, -37.069, 103.492, 142.458, 53.056, -28.988, -355]
  MoveL 4863 to (49.87, 40.63, -275.65) mm, rotated rx 42.04 ry 15.1 rz -114.75 deg; joints [-19.562, -37.037, 103.475, 142.465, 53.068, -29, -355]
  MoveL 4864 to (50.39, 40.68, -275.65) mm, rotated rx 42.04 ry 15.1 rz -114.75 deg; joints [-19.561, -37.004, 103.458, 142.474, 53.08, -29.012, -355]
  MoveL 4865 to (51.08, 40.75, -275.62) mm, rotated rx 42.04 ry 15.1 rz -114.75 deg; joints [-19.558, -36.961, 103.435, 142.486, 53.095, -29.028, -355]
  MoveL 4866 to (51.74, 40.82, -275.59) mm, rotated rx 42.04 ry 15.1 rz -114.75 deg; joints [-19.556, -36.919, 103.412, 142.497, 53.11, -29.044, -355]
  MoveL 4867 to (52.34, 40.88, -275.58) mm, rotated rx 42.04 ry 15.1 rz -114.75 deg; joints [-19.555, -36.882, 103.392, 142.507, 53.123, -29.058, -355]
  MoveL 4868 to (52.81, 40.9, -275.62) mm, rotated rx 42.04 ry 15.1 rz -114.75 deg; joints [-19.556, -36.853, 103.377, 142.512, 53.135, -29.068, -355]
  MoveL 4869 to (53.22, 40.9, -275.68) mm, rotated rx 42.04 ry 15.1 rz -114.75 deg; joints [-19.557, -36.827, 103.365, 142.516, 53.146, -29.078, -355]
  MoveL 4870 to (53.63, 40.91, -275.73) mm, rotated rx 42.04 ry 15.1 rz -114.75 deg; joints [-19.559, -36.802, 103.352, 142.52, 53.156, -29.087, -355]
  MoveL 4871 to (54.07, 40.93, -275.77) mm, rotated rx 42.04 ry 15.1 rz -114.75 deg; joints [-19.56, -36.774, 103.338, 142.525, 53.167, -29.097, -355]
  MoveL 4872 to (55.64, 41.06, -275.77) mm, rotated rx 42.04 ry 15.1 rz -114.75 deg; joints [-19.557, -36.676, 103.286, 142.549, 53.203, -29.133, -355]
  MoveL 4873 to (58.53, 41.08, -276.15) mm, rotated rx 42.04 ry 15.1 rz -114.75 deg; joints [-19.569, -36.497, 103.199, 142.578, 53.279, -29.198, -355]
  MoveL 4874 to (59.77, 40.9, -276.62) mm, rotated rx 42.04 ry 15.1 rz -114.75 deg; joints [-19.587, -36.423, 103.171, 142.578, 53.319, -29.225, -355]
  MoveL 4875 to (60.87, 40.59, -277.28) mm, rotated rx 42.04 ry 15.1 rz -114.75 deg; joints [-19.613, -36.359, 103.152, 142.567, 53.362, -29.249, -355]
  MoveL 4876 to (61.83, 40.16, -278.12) mm, rotated rx 42.04 ry 15.1 rz -114.75 deg; joints [-19.648, -36.305, 103.144, 142.548, 53.406, -29.27, -355]
  MoveL 4877 to (62.66, 39.6, -279.16) mm, rotated rx 42.04 ry 15.1 rz -114.75 deg; joints [-19.692, -36.262, 103.145, 142.518, 53.452, -29.287, -355]
  MoveL 4878 to (63.91, 38.11, -281.8) mm, rotated rx 42.04 ry 15.1 rz -114.75 deg; joints [-19.803, -36.205, 103.178, 142.43, 53.55, -29.312, -355]
  MoveL 4879 to (64.37, 36.59, -284.43) mm, rotated rx 42.04 ry 15.1 rz -114.75 deg; joints [-19.916, -36.196, 103.233, 142.329, 53.628, -29.317, -355]
  MoveL 4880 to (64.21, 35.99, -285.47) mm, rotated rx 42.04 ry 15.1 rz -114.75 deg; joints [-19.961, -36.213, 103.263, 142.284, 53.649, -29.31, -355]
  MoveL 4881 to (63.79, 35.51, -286.32) mm, rotated rx 42.04 ry 15.1 rz -114.75 deg; joints [-19.998, -36.244, 103.295, 142.242, 53.658, -29.297, -355]
  MoveL 4882 to (63.11, 35.15, -286.98) mm, rotated rx 42.04 ry 15.1 rz -114.75 deg; joints [-20.026, -36.29, 103.329, 142.204, 53.656, -29.277, -355]
  MoveL 4883 to (62.17, 34.89, -287.45) mm, rotated rx 42.04 ry 15.1 rz -114.75 deg; joints [-20.047, -36.349, 103.365, 142.169, 53.642, -29.25, -355]
  MoveL 4884 to (60.97, 34.75, -287.73) mm, rotated rx 42.04 ry 15.1 rz -114.75 deg; joints [-20.06, -36.423, 103.402, 142.137, 53.616, -29.218, -355]
  MoveL 4885 to (59.51, 34.72, -287.82) mm, rotated rx 42.04 ry 15.1 rz -114.75 deg; joints [-20.065, -36.512, 103.441, 142.109, 53.578, -29.178, -355]
  MoveL 4886 to (58.99, 34.73, -287.82) mm, rotated rx 42.04 ry 15.1 rz -114.75 deg; joints [-20.066, -36.543, 103.454, 142.101, 53.564, -29.164, -355]
  MoveL 4887 to (58.52, 34.75, -287.8) mm, rotated rx 42.04 ry 15.1 rz -114.75 deg; joints [-20.065, -36.571, 103.466, 142.094, 53.55, -29.151, -355]
  MoveL 4888 to (58.12, 34.78, -287.76) mm, rotated rx 42.04 ry 15.1 rz -114.75 deg; joints [-20.063, -36.595, 103.475, 142.089, 53.538, -29.141, -355]
  MoveL 4889 to (57.73, 34.82, -287.7) mm, rotated rx 42.04 ry 15.1 rz -114.75 deg; joints [-20.061, -36.618, 103.483, 142.085, 53.526, -29.13, -355]
  MoveL 4890 to (57.3, 34.85, -287.66) mm, rotated rx 42.04 ry 15.1 rz -114.75 deg; joints [-20.06, -36.644, 103.493, 142.079, 53.513, -29.119, -355]
  MoveL 4891 to (56.81, 34.87, -287.63) mm, rotated rx 42.04 ry 15.1 rz -114.75 deg; joints [-20.059, -36.673, 103.505, 142.072, 53.499, -29.106, -355]
  MoveL 4892 to (56.29, 34.88, -287.63) mm, rotated rx 42.04 ry 15.1 rz -114.75 deg; joints [-20.059, -36.704, 103.518, 142.063, 53.485, -29.091, -355]
  MoveL 4893 to (55.82, 34.89, -287.61) mm, rotated rx 42.04 ry 15.1 rz -114.75 deg; joints [-20.059, -36.732, 103.529, 142.056, 53.472, -29.079, -355]
  MoveL 4894 to (55.42, 34.91, -287.56) mm, rotated rx 42.04 ry 15.1 rz -114.75 deg; joints [-20.057, -36.757, 103.539, 142.052, 53.46, -29.069, -355]
  MoveL 4895 to (55.03, 34.94, -287.5) mm, rotated rx 42.04 ry 15.1 rz -114.75 deg; joints [-20.055, -36.78, 103.548, 142.048, 53.448, -29.059, -355]
  MoveL 4896 to (54.6, 34.96, -287.45) mm, rotated rx 42.04 ry 15.1 rz -114.75 deg; joints [-20.053, -36.806, 103.559, 142.043, 53.436, -29.047, -355]
  MoveL 4897 to (54.11, 34.98, -287.43) mm, rotated rx 42.04 ry 15.1 rz -114.75 deg; joints [-20.053, -36.835, 103.571, 142.036, 53.422, -29.034, -355]
  MoveL 4898 to (53.58, 34.99, -287.43) mm, rotated rx 42.04 ry 15.1 rz -114.75 deg; joints [-20.053, -36.867, 103.583, 142.027, 53.407, -29.02, -355]
  MoveL 4899 to (52.6, 35.08, -287.41) mm, rotated rx 42.04 ry 15.1 rz -114.75 deg; joints [-20.052, -36.924, 103.602, 142.01, 53.377, -28.991, -355]
  MoveC 4900 to (51.23, 35.24, -287.41) mm, rotated rx 42.04 ry 15.1 rz -114.75 deg; joints [-20.052, -37.002, 103.623, 141.984, 53.332, -28.947, -355] to (49.85, 35.23, -287.41) mm, rotated rx 42.04 ry 15.1 rz -114.75 deg; joints [-20.053, -37.085, 103.659, 141.961, 53.295, -28.91, -355]
  MoveL 4901 to (49.85, 35.23, -287.4) mm, rotated rx 42.04 ry 15.1 rz -114.75 deg; joints [-20.053, -37.085, 103.659, 141.962, 53.295, -28.911, -355]
  MoveL 4902 to (49.19, 35.29, -287.38) mm, rotated rx 42.04 ry 15.1 rz -114.75 deg; joints [-20.052, -37.124, 103.672, 141.951, 53.275, -28.891, -355]
  MoveL 4903 to (48.63, 35.39, -287.35) mm, rotated rx 42.04 ry 15.1 rz -114.75 deg; joints [-20.05, -37.155, 103.678, 141.941, 53.254, -28.872, -355]
  MoveL 4904 to (48.35, 35.51, -287.26) mm, rotated rx 42.04 ry 15.1 rz -114.75 deg; joints [-20.046, -37.169, 103.678, 141.939, 53.241, -28.863, -355]
  MoveL 4905 to (48.41, 35.54, -287.06) mm, rotated rx 42.04 ry 15.1 rz -114.75 deg; joints [-20.038, -37.167, 103.678, 141.949, 53.242, -28.868, -355]
  MoveL 4906 to (48.82, 35.46, -286.75) mm, rotated rx 42.04 ry 15.1 rz -114.75 deg; joints [-20.027, -37.147, 103.683, 141.973, 53.258, -28.891, -355]
  MoveL 4907 to (49.09, 35.73, -286.13) mm, rotated rx 42.04 ry 15.1 rz -114.75 deg; joints [-20.001, -37.129, 103.667, 142.005, 53.254, -28.903, -355]
  MoveL 4908 to (47.36, 36.8, -286.12) mm, rotated rx 42.04 ry 15.1 rz -114.75 deg; joints [-19.991, -37.202, 103.619, 141.96, 53.156, -28.813, -355]
  MoveL 4909 to (45.59, 38, -286.06) mm, rotated rx 42.04 ry 15.1 rz -114.75 deg; joints [-19.978, -37.275, 103.562, 141.914, 53.05, -28.718, -355]
  MoveL 4910 to (43.73, 39.31, -285.94) mm, rotated rx 42.04 ry 15.1 rz -114.75 deg; joints [-19.962, -37.35, 103.498, 141.869, 52.937, -28.618, -355]
  MoveL 4911 to (41.9, 40.6, -285.84) mm, rotated rx 42.04 ry 15.1 rz -114.75 deg; joints [-19.947, -37.423, 103.435, 141.823, 52.826, -28.518, -355]
  MoveL 4912 to (40.14, 41.84, -285.67) mm, rotated rx 42.04 ry 15.1 rz -114.75 deg; joints [-19.929, -37.494, 103.375, 141.782, 52.719, -28.424, -355]
  MoveL 4913 to (38.56, 42.97, -285.52) mm, rotated rx 42.04 ry 15.1 rz -114.75 deg; joints [-19.914, -37.557, 103.32, 141.744, 52.623, -28.338, -355]
  MoveL 4914 to (36.86, 44.15, -285.47) mm, rotated rx 42.04 ry 15.1 rz -114.75 deg; joints [-19.901, -37.624, 103.26, 141.698, 52.52, -28.245, -355]
  MoveL 4915 to (35.1, 45.39, -285.4) mm, rotated rx 42.04 ry 15.1 rz -114.75 deg; joints [-19.888, -37.694, 103.198, 141.651, 52.413, -28.147, -355]
  MoveL 4916 to (33.17, 46.74, -285.25) mm, rotated rx 42.04 ry 15.1 rz -114.75 deg; joints [-19.87, -37.77, 103.131, 141.603, 52.296, -28.042, -355]
  MoveL 4917 to (31.63, 47.82, -285.13) mm, rotated rx 42.04 ry 15.1 rz -114.75 deg; joints [-19.856, -37.83, 103.077, 141.564, 52.203, -27.958, -355]
  MoveL 4918 to (29.67, 49.18, -284.92) mm, rotated rx 42.04 ry 15.1 rz -114.75 deg; joints [-19.836, -37.908, 103.01, 141.518, 52.084, -27.852, -355]
  MoveL 4919 to (28.13, 50.25, -284.8) mm, rotated rx 42.04 ry 15.1 rz -114.75 deg; joints [-19.823, -37.969, 102.957, 141.478, 51.991, -27.768, -355]
  MoveL 4920 to (26.37, 51.46, -284.64) mm, rotated rx 42.04 ry 15.1 rz -114.75 deg; joints [-19.806, -38.038, 102.896, 141.434, 51.886, -27.672, -355]
  MoveL 4921 to (24.41, 52.82, -284.59) mm, rotated rx 42.04 ry 15.1 rz -114.75 deg; joints [-19.792, -38.113, 102.825, 141.378, 51.767, -27.562, -355]
  MoveL 4922 to (22.86, 53.89, -284.48) mm, rotated rx 42.04 ry 15.1 rz -114.75 deg; joints [-19.779, -38.173, 102.77, 141.338, 51.674, -27.476, -355]
  MoveL 4923 to (21.1, 55.1, -284.32) mm, rotated rx 42.04 ry 15.1 rz -114.75 deg; joints [-19.762, -38.242, 102.71, 141.293, 51.569, -27.38, -355]
  MoveL 4924 to (19.14, 56.45, -284.27) mm, rotated rx 42.04 ry 15.1 rz -114.75 deg; joints [-19.748, -38.316, 102.637, 141.236, 51.451, -27.269, -355]
  MoveL 4925 to (17.59, 57.52, -284.15) mm, rotated rx 42.04 ry 15.1 rz -114.75 deg; joints [-19.735, -38.376, 102.582, 141.194, 51.358, -27.183, -355]
  MoveL 4926 to (15.75, 58.77, -284.05) mm, rotated rx 42.04 ry 15.1 rz -114.75 deg; joints [-19.72, -38.446, 102.517, 141.143, 51.248, -27.08, -355]
  MoveL 4927 to (13.92, 60.03, -283.98) mm, rotated rx 42.04 ry 15.1 rz -114.75 deg; joints [-19.707, -38.515, 102.449, 141.09, 51.137, -26.976, -355]
  MoveL 4928 to (12.35, 61.07, -283.8) mm, rotated rx 42.04 ry 15.1 rz -114.75 deg; joints [-19.691, -38.577, 102.397, 141.051, 51.045, -26.891, -355]
  MoveL 4929 to (10.89, 62, -283.55) mm, rotated rx 42.04 ry 15.1 rz -114.75 deg; joints [-19.674, -38.635, 102.354, 141.02, 50.961, -26.816, -355]
  MoveL 4930 to (9.5, 62.85, -283.2) mm, rotated rx 42.04 ry 15.1 rz -114.75 deg; joints [-19.653, -38.693, 102.319, 140.996, 50.883, -26.75, -355]
  MoveL 4931 to (10.45, 61.68, -282.51) mm, rotated rx 42.04 ry 15.1 rz -114.75 deg; joints [-19.639, -38.681, 102.417, 141.069, 50.965, -26.846, -355]
  MoveL 4932 to (10.29, 61.84, -282.5) mm, rotated rx 42.04 ry 15.1 rz -114.75 deg; joints [-19.637, -38.686, 102.407, 141.064, 50.953, -26.835, -355]
  MoveL 4933 to (10.11, 62.08, -282.49) mm, rotated rx 42.04 ry 15.1 rz -114.75 deg; joints [-19.635, -38.689, 102.39, 141.057, 50.937, -26.82, -355]
  MoveL 4934 to (9.89, 62.49, -282.46) mm, rotated rx 42.04 ry 15.1 rz -114.75 deg; joints [-19.63, -38.689, 102.36, 141.047, 50.912, -26.797, -355]
  MoveL 4935 to (9.66, 62.97, -282.42) mm, rotated rx 42.04 ry 15.1 rz -114.75 deg; joints [-19.624, -38.688, 102.324, 141.036, 50.883, -26.771, -355]
  MoveL 4936 to (9.41, 63.53, -282.38) mm, rotated rx 42.04 ry 15.1 rz -114.75 deg; joints [-19.617, -38.685, 102.281, 141.023, 50.849, -26.742, -355]
  MoveL 4937 to (8.45, 65.97, -282.38) mm, rotated rx 42.04 ry 15.1 rz -114.75 deg; joints [-19.594, -38.664, 102.086, 140.962, 50.708, -26.612, -355]
  MoveL 4938 to (8.22, 66.53, -282.35) mm, rotated rx 42.04 ry 15.1 rz -114.75 deg; joints [-19.587, -38.66, 102.042, 140.949, 50.675, -26.582, -355]
  MoveL 4939 to (7.94, 67.16, -282.29) mm, rotated rx 42.04 ry 15.1 rz -114.75 deg; joints [-19.579, -38.657, 101.994, 140.935, 50.638, -26.549, -355]
  MoveL 4940 to (7.69, 67.74, -282.26) mm, rotated rx 42.04 ry 15.1 rz -114.75 deg; joints [-19.572, -38.653, 101.949, 140.922, 50.604, -26.518, -355]
  MoveL 4941 to (7.5, 68.22, -282.26) mm, rotated rx 42.04 ry 15.1 rz -114.75 deg; joints [-19.568, -38.648, 101.91, 140.909, 50.576, -26.492, -355]
  MoveL 4942 to (7.32, 68.68, -282.25) mm, rotated rx 42.04 ry 15.1 rz -114.75 deg; joints [-19.563, -38.644, 101.874, 140.898, 50.55, -26.468, -355]
  MoveL 4943 to (7.13, 69.17, -282.25) mm, rotated rx 42.04 ry 15.1 rz -114.75 deg; joints [-19.559, -38.64, 101.834, 140.885, 50.522, -26.442, -355]
  MoveL 4944 to (6.94, 69.65, -282.24) mm, rotated rx 42.04 ry 15.1 rz -114.75 deg; joints [-19.554, -38.635, 101.796, 140.873, 50.494, -26.416, -355]
  MoveL 4945 to (6.76, 70.09, -282.22) mm, rotated rx 42.04 ry 15.1 rz -114.75 deg; joints [-19.549, -38.632, 101.761, 140.863, 50.468, -26.392, -355]
  MoveL 4946 to (6.57, 70.52, -282.17) mm, rotated rx 42.04 ry 15.1 rz -114.75 deg; joints [-19.543, -38.63, 101.729, 140.854, 50.443, -26.37, -355]
  MoveL 4947 to (6.38, 70.98, -282.15) mm, rotated rx 42.04 ry 15.1 rz -114.75 deg; joints [-19.538, -38.626, 101.692, 140.843, 50.416, -26.346, -355]
  MoveL 4948 to (6.19, 71.47, -282.15) mm, rotated rx 42.04 ry 15.1 rz -114.75 deg; joints [-19.533, -38.622, 101.653, 140.83, 50.388, -26.319, -355]
  MoveL 4949 to (5.8, 72.45, -282.15) mm, rotated rx 42.04 ry 15.1 rz -114.75 deg; joints [-19.524, -38.612, 101.574, 140.805, 50.331, -26.267, -355]
  Set speed (1000.0 mm/s)
  MoveL 4950 to (3.92, 93.98, -282.15) mm, rotated rx 42.04 ry 15.1 rz -114.75 deg; joints [-19.319, -38.009, 99.677, 140.355, 49.271, -25.287, -355]
  Print: /'Flow1'
  Set speed (1000.0 mm/s)
  MoveL 4951 to (-115.82, -27.66, -72.15) mm, rotated rx -9.61 ry -16.54 rz -54.03 deg; joints [-7.663, -63.141, 109.635, 206.123, 32.592, -123.586, -415]
  Set speed (1000.0 mm/s)
  MoveL 4952 to (-75.15, -46.62, -72.15) mm, rotated rx -9.61 ry -16.54 rz -54.03 deg; joints [-7.768, -65.146, 113.572, 204.695, 34.306, -121.967, -415]
  Set speed (100.0 mm/s)
  MoveL 4953 to (-9.2, -77.37, -72.15) mm, rotated rx -9.61 ry -16.54 rz -54.03 deg; joints [-7.953, -68.3, 119.737, 202.712, 37.017, -119.702, -415]
  MoveL 4954 to (-8.97, -77.84, -72.15) mm, rotated rx -9.61 ry -16.54 rz -54.03 deg; joints [-7.954, -68.336, 119.771, 202.712, 37.014, -119.703, -415]
  MoveL 4955 to (-8.63, -78.39, -72.05) mm, rotated rx -9.61 ry -16.54 rz -54.03 deg; joints [-7.951, -68.379, 119.815, 202.716, 37.015, -119.705, -415]
  MoveL 4956 to (-8.33, -78.9, -72) mm, rotated rx -9.61 ry -16.54 rz -54.03 deg; joints [-7.95, -68.419, 119.854, 202.718, 37.015, -119.707, -415]
  MoveL 4957 to (-8.06, -79.4, -71.98) mm, rotated rx -9.61 ry -16.54 rz -54.03 deg; joints [-7.95, -68.458, 119.89, 202.719, 37.012, -119.708, -415]
  MoveL 4958 to (-6.41, -82.67, -71.98) mm, rotated rx -9.61 ry -16.54 rz -54.03 deg; joints [-7.958, -68.712, 120.122, 202.718, 36.99, -119.715, -415]
  MoveL 4959 to (-5.81, -83.99, -72.06) mm, rotated rx -9.61 ry -16.54 rz -54.03 deg; joints [-7.965, -68.813, 120.209, 202.714, 36.976, -119.717, -415]
  MoveL 4960 to (-5.44, -85.12, -72.33) mm, rotated rx -9.61 ry -16.54 rz -54.03 deg; joints [-7.98, -68.897, 120.272, 202.704, 36.952, -119.717, -415]
  MoveL 4961 to (-5.3, -86.06, -72.77) mm, rotated rx -9.61 ry -16.54 rz -54.03 deg; joints [-8.001, -68.964, 120.309, 202.685, 36.921, -119.715, -415]
  MoveL 4962 to (-5.32, -86.45, -73.06) mm, rotated rx -9.61 ry -16.54 rz -54.03 deg; joints [-8.014, -68.991, 120.319, 202.674, 36.901, -119.714, -415]
  MoveL 4963 to (-5.4, -86.8, -73.4) mm, rotated rx -9.61 ry -16.54 rz -54.03 deg; joints [-8.029, -69.013, 120.322, 202.66, 36.88, -119.712, -415]
  MoveL 4964 to (-5.73, -87.36, -74.19) mm, rotated rx -9.61 ry -16.54 rz -54.03 deg; joints [-8.065, -69.045, 120.31, 202.627, 36.831, -119.705, -415]
  MoveL 4965 to (-6.29, -87.72, -75.17) mm, rotated rx -9.61 ry -16.54 rz -54.03 deg; joints [-8.108, -69.059, 120.273, 202.588, 36.773, -119.697, -415]
  MoveL 4966 to (-8.11, -87.87, -77.66) mm, rotated rx -9.61 ry -16.54 rz -54.03 deg; joints [-8.214, -69.036, 120.125, 202.486, 36.632, -119.674, -415]
  MoveL 4967 to (-10.25, -87.29, -80.14) mm, rotated rx -9.61 ry -16.54 rz -54.03 deg; joints [-8.318, -68.956, 119.929, 202.383, 36.5, -119.647, -415]
  MoveL 4968 to (-12.1, -86.03, -81.91) mm, rotated rx -9.61 ry -16.54 rz -54.03 deg; joints [-8.391, -68.835, 119.738, 202.306, 36.418, -119.621, -415]
  MoveL 4969 to (-12.91, -85.14, -82.54) mm, rotated rx -9.61 ry -16.54 rz -54.03 deg; joints [-8.415, -68.759, 119.644, 202.277, 36.396, -119.608, -415]
  MoveL 4970 to (-13.64, -84.08, -82.98) mm, rotated rx -9.61 ry -16.54 rz -54.03 deg; joints [-8.431, -68.672, 119.551, 202.255, 36.386, -119.596, -415]
  MoveL 4971 to (-14.89, -81.45, -83.33) mm, rotated rx -9.61 ry -16.54 rz -54.03 deg; joints [-8.44, -68.468, 119.37, 202.23, 36.405, -119.574, -415]
  MoveL 4972 to (-15.99, -78.5, -83.34) mm, rotated rx -9.61 ry -16.54 rz -54.03 deg; joints [-8.433, -68.246, 119.192, 202.218, 36.447, -119.552, -415]
  MoveL 4973 to (-16.17, -78.04, -83.36) mm, rotated rx -9.61 ry -16.54 rz -54.03 deg; joints [-8.432, -68.212, 119.163, 202.216, 36.453, -119.549, -415]
  MoveL 4974 to (-16.35, -77.62, -83.4) mm, rotated rx -9.61 ry -16.54 rz -54.03 deg; joints [-8.433, -68.18, 119.135, 202.213, 36.457, -119.545, -415]
  MoveL 4975 to (-16.54, -77.25, -83.46) mm, rotated rx -9.61 ry -16.54 rz -54.03 deg; joints [-8.435, -68.151, 119.109, 202.209, 36.459, -119.542, -415]
  MoveL 4976 to (-16.72, -76.84, -83.51) mm, rotated rx -9.61 ry -16.54 rz -54.03 deg; joints [-8.436, -68.119, 119.081, 202.205, 36.462, -119.539, -415]
  MoveL 4977 to (-16.92, -76.33, -83.54) mm, rotated rx -9.61 ry -16.54 rz -54.03 deg; joints [-8.436, -68.081, 119.049, 202.202, 36.468, -119.535, -415]
  MoveL 4978 to (-17.17, -75.73, -83.57) mm, rotated rx -9.61 ry -16.54 rz -54.03 deg; joints [-8.436, -68.035, 119.011, 202.198, 36.474, -119.53, -415]
  MoveL 4979 to (-17.39, -75.22, -83.63) mm, rotated rx -9.61 ry -16.54 rz -54.03 deg; joints [-8.437, -67.996, 118.977, 202.194, 36.479, -119.526, -415]
  MoveL 4980 to (-17.59, -74.82, -83.71) mm, rotated rx -9.61 ry -16.54 rz -54.03 deg; joints [-8.439, -67.965, 118.948, 202.189, 36.481, -119.522, -415]
  MoveL 4981 to (-17.77, -74.42, -83.76) mm, rotated rx -9.61 ry -16.54 rz -54.03 deg; joints [-8.44, -67.935, 118.922, 202.185, 36.484, -119.518, -415]
  MoveL 4982 to (-17.95, -73.98, -83.78) mm, rotated rx -9.61 ry -16.54 rz -54.03 deg; joints [-8.44, -67.901, 118.893, 202.183, 36.489, -119.515, -415]
  MoveL 4983 to (-18.13, -73.49, -83.78) mm, rotated rx -9.61 ry -16.54 rz -54.03 deg; joints [-8.439, -67.864, 118.864, 202.181, 36.496, -119.512, -415]
  MoveL 4984 to (-18.32, -72.98, -83.78) mm, rotated rx -9.61 ry -16.54 rz -54.03 deg; joints [-8.438, -67.826, 118.833, 202.179, 36.503, -119.508, -415]
  MoveL 4985 to (-18.53, -72.45, -83.79) mm, rotated rx -9.61 ry -16.54 rz -54.03 deg; joints [-8.437, -67.786, 118.799, 202.177, 36.509, -119.505, -415]
  MoveL 4986 to (-18.79, -71.84, -83.82) mm, rotated rx -9.61 ry -16.54 rz -54.03 deg; joints [-8.437, -67.74, 118.759, 202.174, 36.515, -119.501, -415]
  MoveL 4987 to (-19.05, -71.31, -83.89) mm, rotated rx -9.61 ry -16.54 rz -54.03 deg; joints [-8.438, -67.699, 118.721, 202.17, 36.517, -119.498, -415]
  MoveL 4988 to (-19.28, -70.92, -83.99) mm, rotated rx -9.61 ry -16.54 rz -54.03 deg; joints [-8.442, -67.668, 118.69, 202.165, 36.517, -119.494, -415]
  MoveL 4989 to (-19.27, -70.91, -84.23) mm, rotated rx -9.61 ry -16.54 rz -54.03 deg; joints [-8.452, -67.667, 118.69, 202.148, 36.514, -119.484, -415]
  MoveL 4990 to (-19.02, -71.22, -84.58) mm, rotated rx -9.61 ry -16.54 rz -54.03 deg; joints [-8.469, -67.691, 118.717, 202.121, 36.513, -119.466, -415]
  MoveL 4991 to (-19.23, -72.04, -85.55) mm, rotated rx -9.61 ry -16.54 rz -54.03 deg; joints [-8.512, -67.742, 118.722, 202.077, 36.461, -119.453, -415]
  MoveL 4992 to (-20.95, -70.79, -85.55) mm, rotated rx -9.61 ry -16.54 rz -54.03 deg; joints [-8.505, -67.629, 118.548, 202.118, 36.405, -119.498, -415]
  MoveL 4993 to (-22.83, -69.48, -85.68) mm, rotated rx -9.61 ry -16.54 rz -54.03 deg; joints [-8.504, -67.51, 118.36, 202.156, 36.342, -119.543, -415]
  MoveL 4994 to (-24.6, -68.21, -85.74) mm, rotated rx -9.61 ry -16.54 rz -54.03 deg; joints [-8.5, -67.395, 118.181, 202.195, 36.284, -119.588, -415]
  MoveL 4995 to (-26.34, -66.98, -85.87) mm, rotated rx -9.61 ry -16.54 rz -54.03 deg; joints [-8.499, -67.284, 118.006, 202.229, 36.225, -119.629, -415]
  MoveL 4996 to (-28.09, -65.75, -86.02) mm, rotated rx -9.61 ry -16.54 rz -54.03 deg; joints [-8.499, -67.172, 117.83, 202.262, 36.165, -119.67, -415]
  MoveL 4997 to (-29.82, -64.51, -86.15) mm, rotated rx -9.61 ry -16.54 rz -54.03 deg; joints [-8.498, -67.06, 117.654, 202.296, 36.107, -119.712, -415]
  MoveL 4998 to (-31.56, -63.27, -86.35) mm, rotated rx -9.61 ry -16.54 rz -54.03 deg; joints [-8.501, -66.947, 117.477, 202.326, 36.046, -119.751, -415]
  MoveL 4999 to (-33.29, -62.04, -86.47) mm, rotated rx -9.61 ry -16.54 rz -54.03 deg; joints [-8.5, -66.835, 117.301, 202.361, 35.987, -119.794, -415]
  MoveL 5000 to (-35.03, -60.78, -86.53) mm, rotated rx -9.61 ry -16.54 rz -54.03 deg; joints [-8.496, -66.722, 117.124, 202.401, 35.929, -119.839, -415]
  MoveL 5001 to (-36.78, -59.52, -86.67) mm, rotated rx -9.61 ry -16.54 rz -54.03 deg; joints [-8.495, -66.608, 116.946, 202.436, 35.87, -119.882, -415]
  MoveL 5002 to (-38.59, -58.22, -86.85) mm, rotated rx -9.61 ry -16.54 rz -54.03 deg; joints [-8.496, -66.491, 116.761, 202.47, 35.807, -119.924, -415]
  MoveL 5003 to (-40.39, -56.91, -87.03) mm, rotated rx -9.61 ry -16.54 rz -54.03 deg; joints [-8.498, -66.373, 116.576, 202.503, 35.745, -119.967, -415]
  MoveL 5004 to (-41.91, -55.81, -87.27) mm, rotated rx -9.61 ry -16.54 rz -54.03 deg; joints [-8.502, -66.273, 116.419, 202.526, 35.692, -119.999, -415]
  MoveL 5005 to (-44.06, -54.24, -87.38) mm, rotated rx -9.61 ry -16.54 rz -54.03 deg; joints [-8.499, -66.131, 116.198, 202.574, 35.619, -120.055, -415]
  Set speed (1000.0 mm/s)
  MoveL 5006 to (-85.12, -35.09, -87.38) mm, rotated rx -9.61 ry -16.54 rz -54.03 deg; joints [-8.367, -64.157, 112.299, 203.882, 33.884, -121.526, -415]
  Set speed (1000.0 mm/s)
  MoveL 5007 to (-82.7, -29.9, -99.26) mm, rotated rx -9.61 ry -16.54 rz -54.03 deg; joints [-8.859, -63.812, 112.239, 202.9, 34.015, -120.785, -415]
  Set speed (100.0 mm/s)
  MoveL 5008 to (-56.7, -42.02, -99.26) mm, rotated rx -9.61 ry -16.54 rz -54.03 deg; joints [-8.952, -65.059, 114.72, 202.065, 35.132, -119.855, -415]
  MoveL 5009 to (-55.46, -43.21, -99.02) mm, rotated rx -9.61 ry -16.54 rz -54.03 deg; joints [-8.947, -65.16, 114.859, 202.052, 35.169, -119.835, -415]
  MoveL 5010 to (-53.98, -44.58, -98.95) mm, rotated rx -9.61 ry -16.54 rz -54.03 deg; joints [-8.951, -65.278, 115.023, 202.021, 35.211, -119.801, -415]
  MoveL 5011 to (-52.47, -45.98, -98.81) mm, rotated rx -9.61 ry -16.54 rz -54.03 deg; joints [-8.951, -65.397, 115.19, 201.995, 35.255, -119.77, -415]
  MoveL 5012 to (-50.68, -47.67, -98.67) mm, rotated rx -9.61 ry -16.54 rz -54.03 deg; joints [-8.953, -65.54, 115.388, 201.963, 35.305, -119.732, -415]
  MoveL 5013 to (-49.11, -49.12, -98.67) mm, rotated rx -9.61 ry -16.54 rz -54.03 deg; joints [-8.96, -65.664, 115.56, 201.926, 35.349, -119.693, -415]
  MoveL 5014 to (-47.38, -50.72, -98.51) mm, rotated rx -9.61 ry -16.54 rz -54.03 deg; joints [-8.961, -65.8, 115.751, 201.896, 35.399, -119.657, -415]
  MoveL 5015 to (-45.92, -52.07, -98.33) mm, rotated rx -9.61 ry -16.54 rz -54.03 deg; joints [-8.96, -65.916, 115.912, 201.875, 35.441, -119.63, -415]
  MoveL 5016 to (-44.42, -53.47, -98.24) mm, rotated rx -9.61 ry -16.54 rz -54.03 deg; joints [-8.962, -66.035, 116.076, 201.847, 35.482, -119.598, -415]
  MoveL 5017 to (-42.85, -54.91, -98.02) mm, rotated rx -9.61 ry -16.54 rz -54.03 deg; joints [-8.96, -66.159, 116.249, 201.825, 35.528, -119.57, -415]
  MoveL 5018 to (-41.29, -56.34, -97.86) mm, rotated rx -9.61 ry -16.54 rz -54.03 deg; joints [-8.96, -66.282, 116.419, 201.8, 35.572, -119.539, -415]
  MoveL 5019 to (-39.73, -57.77, -97.75) mm, rotated rx -9.61 ry -16.54 rz -54.03 deg; joints [-8.962, -66.404, 116.589, 201.772, 35.616, -119.507, -415]
  MoveL 5020 to (-38.15, -59.21, -97.58) mm, rotated rx -9.61 ry -16.54 rz -54.03 deg; joints [-8.962, -66.528, 116.761, 201.748, 35.661, -119.476, -415]
  MoveL 5021 to (-36.58, -60.64, -97.44) mm, rotated rx -9.61 ry -16.54 rz -54.03 deg; joints [-8.963, -66.651, 116.931, 201.722, 35.705, -119.445, -415]
  MoveL 5022 to (-34.97, -62.11, -97.38) mm, rotated rx -9.61 ry -16.54 rz -54.03 deg; joints [-8.967, -66.777, 117.105, 201.69, 35.748, -119.41, -415]
  MoveL 5023 to (-33.38, -63.53, -97.17) mm, rotated rx -9.61 ry -16.54 rz -54.03 deg; joints [-8.965, -66.9, 117.277, 201.668, 35.794, -119.381, -415]
  MoveL 5024 to (-31.81, -64.95, -97.04) mm, rotated rx -9.61 ry -16.54 rz -54.03 deg; joints [-8.967, -67.022, 117.447, 201.642, 35.838, -119.35, -415]
  MoveL 5025 to (-30.2, -66.4, -96.92) mm, rotated rx -9.61 ry -16.54 rz -54.03 deg; joints [-8.969, -67.147, 117.619, 201.614, 35.882, -119.318, -415]
  MoveL 5026 to (-28.8, -67.49, -96.71) mm, rotated rx -9.61 ry -16.54 rz -54.03 deg; joints [-8.966, -67.244, 117.765, 201.595, 35.927, -119.291, -415]
  MoveL 5027 to (-27.56, -68.28, -96.36) mm, rotated rx -9.61 ry -16.54 rz -54.03 deg; joints [-8.955, -67.319, 117.889, 201.586, 35.976, -119.27, -415]
  MoveL 5028 to (-26.45, -68.76, -95.83) mm, rotated rx -9.61 ry -16.54 rz -54.03 deg; joints [-8.936, -67.371, 117.994, 201.589, 36.029, -119.256, -415]
  MoveL 5029 to (-27.22, -67.43, -94.98) mm, rotated rx -9.61 ry -16.54 rz -54.03 deg; joints [-8.895, -67.27, 117.897, 201.653, 36.042, -119.296, -415]
  MoveL 5030 to (-26.76, -68.08, -94.98) mm, rotated rx -9.61 ry -16.54 rz -54.03 deg; joints [-8.897, -67.323, 117.954, 201.647, 36.046, -119.29, -415]
  MoveL 5031 to (-26.41, -68.69, -94.98) mm, rotated rx -9.61 ry -16.54 rz -54.03 deg; joints [-8.899, -67.37, 118.001, 201.644, 36.045, -119.288, -415]
  MoveL 5032 to (-26.18, -69.29, -94.97) mm, rotated rx -9.61 ry -16.54 rz -54.03 deg; joints [-8.9, -67.415, 118.038, 201.646, 36.038, -119.292, -415]
  MoveL 5033 to (-25.98, -69.92, -94.95) mm, rotated rx -9.61 ry -16.54 rz -54.03 deg; joints [-8.901, -67.462, 118.074, 201.65, 36.028, -119.298, -415]
  MoveL 5034 to (-25.77, -70.66, -94.92) mm, rotated rx -9.61 ry -16.54 rz -54.03 deg; joints [-8.902, -67.516, 118.114, 201.657, 36.015, -119.306, -415]
  MoveL 5035 to (-25.28, -72.7, -94.92) mm, rotated rx -9.61 ry -16.54 rz -54.03 deg; joints [-8.906, -67.664, 118.218, 201.672, 35.972, -119.329, -415]
  MoveL 5036 to (-25.17, -73.13, -94.9) mm, rotated rx -9.61 ry -16.54 rz -54.03 deg; joints [-8.907, -67.696, 118.241, 201.676, 35.964, -119.335, -415]
  MoveL 5037 to (-24.92, -74.15, -94.9) mm, rotated rx -9.61 ry -16.54 rz -54.03 deg; joints [-8.909, -67.77, 118.292, 201.684, 35.942, -119.347, -415]
  MoveL 5038 to (-24.8, -74.64, -94.89) mm, rotated rx -9.61 ry -16.54 rz -54.03 deg; joints [-8.91, -67.806, 118.318, 201.688, 35.932, -119.352, -415]
  MoveL 5039 to (-24.68, -75.11, -94.87) mm, rotated rx -9.61 ry -16.54 rz -54.03 deg; joints [-8.91, -67.841, 118.343, 201.692, 35.923, -119.358, -415]
  MoveL 5040 to (-24.54, -75.57, -94.84) mm, rotated rx -9.61 ry -16.54 rz -54.03 deg; joints [-8.91, -67.875, 118.368, 201.697, 35.915, -119.364, -415]
  MoveL 5041 to (-24.4, -75.98, -94.78) mm, rotated rx -9.61 ry -16.54 rz -54.03 deg; joints [-8.909, -67.906, 118.392, 201.703, 35.909, -119.37, -415]
  MoveL 5042 to (-24.27, -76.44, -94.75) mm, rotated rx -9.61 ry -16.54 rz -54.03 deg; joints [-8.908, -67.939, 118.417, 201.708, 35.901, -119.376, -415]
  MoveL 5043 to (-24.14, -76.91, -94.73) mm, rotated rx -9.61 ry -16.54 rz -54.03 deg; joints [-8.908, -67.974, 118.442, 201.712, 35.892, -119.381, -415]
  MoveL 5044 to (-24.02, -77.41, -94.72) mm, rotated rx -9.61 ry -16.54 rz -54.03 deg; joints [-8.909, -68.01, 118.468, 201.717, 35.882, -119.387, -415]
  MoveL 5045 to (-23.89, -77.88, -94.7) mm, rotated rx -9.61 ry -16.54 rz -54.03 deg; joints [-8.91, -68.045, 118.493, 201.721, 35.873, -119.393, -415]
  MoveL 5046 to (-23.75, -78.34, -94.67) mm, rotated rx -9.61 ry -16.54 rz -54.03 deg; joints [-8.909, -68.079, 118.518, 201.726, 35.865, -119.399, -415]
  MoveL 5047 to (-23.61, -78.75, -94.61) mm, rotated rx -9.61 ry -16.54 rz -54.03 deg; joints [-8.908, -68.11, 118.543, 201.731, 35.859, -119.404, -415]
  MoveL 5048 to (-23.46, -79.18, -94.55) mm, rotated rx -9.61 ry -16.54 rz -54.03 deg; joints [-8.907, -68.143, 118.568, 201.737, 35.853, -119.41, -415]
  MoveL 5049 to (-23.06, -80.57, -94.47) mm, rotated rx -9.61 ry -16.54 rz -54.03 deg; joints [-8.906, -68.245, 118.644, 201.751, 35.828, -119.427, -415]
  MoveL 5050 to (-22.88, -81.73, -94.6) mm, rotated rx -9.61 ry -16.54 rz -54.03 deg; joints [-8.914, -68.328, 118.694, 201.755, 35.796, -119.44, -415]
  MoveL 5051 to (-22.91, -82.67, -94.94) mm, rotated rx -9.61 ry -16.54 rz -54.03 deg; joints [-8.931, -68.392, 118.719, 201.749, 35.756, -119.448, -415]
  MoveL 5052 to (-23.01, -83.06, -95.18) mm, rotated rx -9.61 ry -16.54 rz -54.03 deg; joints [-8.942, -68.416, 118.722, 201.742, 35.733, -119.45, -415]
  MoveL 5053 to (-23.16, -83.39, -95.48) mm, rotated rx -9.61 ry -16.54 rz -54.03 deg; joints [-8.955, -68.436, 118.719, 201.733, 35.709, -119.451, -415]
  MoveL 5054 to (-23.62, -83.9, -96.24) mm, rotated rx -9.61 ry -16.54 rz -54.03 deg; joints [-8.988, -68.461, 118.694, 201.706, 35.655, -119.449, -415]
  MoveL 5055 to (-24.31, -84.18, -97.21) mm, rotated rx -9.61 ry -16.54 rz -54.03 deg; joints [-9.029, -68.466, 118.644, 201.669, 35.593, -119.443, -415]
  MoveL 5056 to (-26.32, -84.09, -99.77) mm, rotated rx -9.61 ry -16.54 rz -54.03 deg; joints [-9.136, -68.419, 118.468, 201.565, 35.449, -119.415, -415]
  MoveL 5057 to (-28.5, -83.24, -102.39) mm, rotated rx -9.61 ry -16.54 rz -54.03 deg; joints [-9.242, -68.314, 118.254, 201.451, 35.322, -119.375, -415]
  MoveL 5058 to (-29.39, -82.56, -103.41) mm, rotated rx -9.61 ry -16.54 rz -54.03 deg; joints [-9.283, -68.249, 118.156, 201.402, 35.281, -119.353, -415]
  MoveL 5059 to (-30.16, -81.72, -104.25) mm, rotated rx -9.61 ry -16.54 rz -54.03 deg; joints [-9.315, -68.176, 118.064, 201.358, 35.257, -119.33, -415]
  MoveL 5060 to (-30.79, -80.72, -104.9) mm, rotated rx -9.61 ry -16.54 rz -54.03 deg; joints [-9.34, -68.094, 117.979, 201.32, 35.248, -119.307, -415]
  MoveL 5061 to (-31.3, -79.55, -105.37) mm, rotated rx -9.61 ry -16.54 rz -54.03 deg; joints [-9.357, -68.004, 117.899, 201.288, 35.254, -119.283, -415]
  MoveL 5062 to (-31.67, -78.22, -105.65) mm, rotated rx -9.61 ry -16.54 rz -54.03 deg; joints [-9.365, -67.905, 117.826, 201.261, 35.276, -119.258, -415]
  MoveL 5063 to (-31.92, -76.73, -105.74) mm, rotated rx -9.61 ry -16.54 rz -54.03 deg; joints [-9.366, -67.798, 117.759, 201.239, 35.313, -119.232, -415]
  MoveL 5064 to (-32.27, -73.59, -105.75) mm, rotated rx -9.61 ry -16.54 rz -54.03 deg; joints [-9.359, -67.576, 117.631, 201.203, 35.402, -119.181, -415]
  MoveL 5065 to (-32.34, -73.04, -105.76) mm, rotated rx -9.61 ry -16.54 rz -54.03 deg; joints [-9.358, -67.537, 117.608, 201.196, 35.417, -119.172, -415]
  MoveL 5066 to (-32.44, -72.42, -105.8) mm, rotated rx -9.61 ry -16.54 rz -54.03 deg; joints [-9.358, -67.493, 117.58, 201.187, 35.432, -119.161, -415]
  MoveL 5067 to (-32.58, -71.68, -105.89) mm, rotated rx -9.61 ry -16.54 rz -54.03 deg; joints [-9.361, -67.439, 117.544, 201.174, 35.449, -119.148, -415]
  MoveL 5068 to (-32.68, -71.07, -105.93) mm, rotated rx -9.61 ry -16.54 rz -54.03 deg; joints [-9.361, -67.395, 117.517, 201.166, 35.464, -119.137, -415]
  MoveL 5069 to (-32.75, -70.53, -105.94) mm, rotated rx -9.61 ry -16.54 rz -54.03 deg; joints [-9.36, -67.357, 117.494, 201.159, 35.478, -119.128, -415]
  MoveL 5070 to (-32.81, -70.02, -105.95) mm, rotated rx -9.61 ry -16.54 rz -54.03 deg; joints [-9.36, -67.321, 117.473, 201.153, 35.492, -119.12, -415]
  MoveL 5071 to (-32.88, -69.57, -105.97) mm, rotated rx -9.61 ry -16.54 rz -54.03 deg; joints [-9.359, -67.289, 117.453, 201.147, 35.504, -119.113, -415]
  MoveL 5072 to (-33.12, -67.53, -105.97) mm, rotated rx -9.61 ry -16.54 rz -54.03 deg; joints [-9.355, -67.145, 117.368, 201.124, 35.56, -119.08, -415]
  MoveL 5073 to (-33.2, -67.02, -106.01) mm, rotated rx -9.61 ry -16.54 rz -54.03 deg; joints [-9.355, -67.109, 117.345, 201.117, 35.572, -119.072, -415]
  MoveL 5074 to (-33.29, -66.56, -106.06) mm, rotated rx -9.61 ry -16.54 rz -54.03 deg; joints [-9.356, -67.075, 117.323, 201.109, 35.582, -119.064, -415]
  MoveL 5075 to (-33.39, -66.11, -106.13) mm, rotated rx -9.61 ry -16.54 rz -54.03 deg; joints [-9.358, -67.042, 117.299, 201.101, 35.591, -119.056, -415]
  MoveL 5076 to (-33.53, -65.64, -106.19) mm, rotated rx -9.61 ry -16.54 rz -54.03 deg; joints [-9.36, -67.008, 117.273, 201.095, 35.598, -119.049, -415]
  MoveL 5077 to (-33.69, -65.11, -106.23) mm, rotated rx -9.61 ry -16.54 rz -54.03 deg; joints [-9.36, -66.969, 117.243, 201.091, 35.606, -119.044, -415]
  MoveL 5078 to (-33.98, -64.51, -106.24) mm, rotated rx -9.61 ry -16.54 rz -54.03 deg; joints [-9.358, -66.923, 117.2, 201.092, 35.61, -119.043, -415]
  MoveL 5079 to (-34.38, -63.84, -106.24) mm, rotated rx -9.61 ry -16.54 rz -54.03 deg; joints [-9.356, -66.871, 117.148, 201.096, 35.61, -119.046, -415]
  MoveL 5080 to (-34.29, -65.78, -107.79) mm, rotated rx -9.61 ry -16.54 rz -54.03 deg; joints [-9.427, -66.999, 117.207, 201.017, 35.529, -119.016, -415]
  MoveL 5081 to (-35.84, -64, -107.92) mm, rotated rx -9.61 ry -16.54 rz -54.03 deg; joints [-9.424, -66.852, 117.027, 201.037, 35.499, -119.039, -415]
  MoveL 5082 to (-37.3, -62.31, -108.03) mm, rotated rx -9.61 ry -16.54 rz -54.03 deg; joints [-9.421, -66.713, 116.857, 201.058, 35.471, -119.061, -415]
  MoveL 5083 to (-38.73, -60.68, -108.19) mm, rotated rx -9.61 ry -16.54 rz -54.03 deg; joints [-9.42, -66.579, 116.692, 201.075, 35.442, -119.082, -415]
  MoveL 5084 to (-40.12, -59.07, -108.3) mm, rotated rx -9.61 ry -16.54 rz -54.03 deg; joints [-9.418, -66.446, 116.529, 201.095, 35.414, -119.103, -415]
  MoveL 5085 to (-41.52, -57.45, -108.41) mm, rotated rx -9.61 ry -16.54 rz -54.03 deg; joints [-9.415, -66.313, 116.365, 201.114, 35.386, -119.125, -415]
  MoveL 5086 to (-42.92, -55.84, -108.63) mm, rotated rx -9.61 ry -16.54 rz -54.03 deg; joints [-9.417, -66.181, 116.201, 201.127, 35.356, -119.143, -415]
  MoveL 5087 to (-44.32, -54.23, -108.86) mm, rotated rx -9.61 ry -16.54 rz -54.03 deg; joints [-9.419, -66.048, 116.036, 201.14, 35.326, -119.16, -415]
  MoveL 5088 to (-45.71, -52.61, -108.97) mm, rotated rx -9.61 ry -16.54 rz -54.03 deg; joints [-9.416, -65.915, 115.872, 201.16, 35.298, -119.182, -415]
  MoveL 5089 to (-47.09, -50.98, -108.97) mm, rotated rx -9.61 ry -16.54 rz -54.03 deg; joints [-9.409, -65.782, 115.71, 201.187, 35.272, -119.209, -415]
  MoveL 5090 to (-48.48, -49.36, -109.08) mm, rotated rx -9.61 ry -16.54 rz -54.03 deg; joints [-9.406, -65.65, 115.546, 201.207, 35.243, -119.231, -415]
  MoveL 5091 to (-49.88, -47.71, -109.29) mm, rotated rx -9.61 ry -16.54 rz -54.03 deg; joints [-9.408, -65.515, 115.379, 201.222, 35.213, -119.25, -415]
  MoveL 5092 to (-51.19, -46.18, -109.47) mm, rotated rx -9.61 ry -16.54 rz -54.03 deg; joints [-9.408, -65.389, 115.223, 201.236, 35.185, -119.268, -415]
  MoveL 5093 to (-52.39, -44.76, -109.68) mm, rotated rx -9.61 ry -16.54 rz -54.03 deg; joints [-9.411, -65.273, 115.079, 201.246, 35.158, -119.282, -415]
  MoveL 5094 to (-53.66, -43.26, -109.77) mm, rotated rx -9.61 ry -16.54 rz -54.03 deg; joints [-9.408, -65.151, 114.928, 201.266, 35.131, -119.304, -415]
  MoveL 5095 to (-55.01, -41.67, -109.79) mm, rotated rx -9.61 ry -16.54 rz -54.03 deg; joints [-9.402, -65.021, 114.767, 201.292, 35.104, -119.331, -415]
  MoveL 5096 to (-56.75, -39.59, -109.88) mm, rotated rx -9.61 ry -16.54 rz -54.03 deg; joints [-9.397, -64.853, 114.558, 201.322, 35.067, -119.361, -415]
  MoveL 5097 to (-58.05, -38.03, -110.1) mm, rotated rx -9.61 ry -16.54 rz -54.03 deg; joints [-9.399, -64.725, 114.4, 201.334, 35.039, -119.378, -415]
  MoveL 5098 to (-59.45, -36.33, -110.3) mm, rotated rx -9.61 ry -16.54 rz -54.03 deg; joints [-9.4, -64.587, 114.23, 201.349, 35.008, -119.398, -415]
  MoveL 5099 to (-60.73, -34.76, -110.58) mm, rotated rx -9.61 ry -16.54 rz -54.03 deg; joints [-9.405, -64.46, 114.073, 201.356, 34.979, -119.411, -415]
  MoveL 5100 to (-62, -33.24, -110.71) mm, rotated rx -9.61 ry -16.54 rz -54.03 deg; joints [-9.404, -64.336, 113.919, 201.374, 34.951, -119.432, -415]
  MoveL 5101 to (-63.36, -31.64, -110.73) mm, rotated rx -9.61 ry -16.54 rz -54.03 deg; joints [-9.397, -64.207, 113.756, 201.402, 34.922, -119.46, -415]
  MoveL 5102 to (-64.46, -30.25, -110.96) mm, rotated rx -9.61 ry -16.54 rz -54.03 deg; joints [-9.401, -64.095, 113.619, 201.409, 34.897, -119.472, -415]
  Set speed (1000.0 mm/s)
  MoveL 5103 to (-88.08, -19.24, -110.96) mm, rotated rx -9.61 ry -16.54 rz -54.03 deg; joints [-9.309, -62.966, 111.351, 202.177, 33.862, -120.32, -415]
  Set speed (1000.0 mm/s)
  MoveL 5104 to (-85.31, -13.32, -122.15) mm, rotated rx -9.61 ry -16.54 rz -54.03 deg; joints [-9.767, -62.572, 111.273, 201.243, 34.045, -119.606, -415]
  Set speed (100.0 mm/s)
  MoveL 5105 to (-67.03, -21.84, -122.15) mm, rotated rx -9.61 ry -16.54 rz -54.03 deg; joints [-9.843, -63.44, 113.032, 200.653, 34.858, -118.961, -415]
  MoveL 5106 to (-65.87, -23.63, -122.15) mm, rotated rx -9.61 ry -16.54 rz -54.03 deg; joints [-9.851, -63.579, 113.188, 200.632, 34.872, -118.942, -415]
  MoveL 5107 to (-64.67, -25.51, -122.05) mm, rotated rx -9.61 ry -16.54 rz -54.03 deg; joints [-9.855, -63.725, 113.35, 200.618, 34.886, -118.929, -415]
  MoveL 5108 to (-63.44, -27.51, -121.75) mm, rotated rx -9.61 ry -16.54 rz -54.03 deg; joints [-9.85, -63.88, 113.52, 200.617, 34.901, -118.924, -415]
  MoveL 5109 to (-62.26, -29.43, -121.41) mm, rotated rx -9.61 ry -16.54 rz -54.03 deg; joints [-9.844, -64.03, 113.683, 200.621, 34.915, -118.923, -415]
  MoveL 5110 to (-61.15, -31.18, -121.22) mm, rotated rx -9.61 ry -16.54 rz -54.03 deg; joints [-9.843, -64.166, 113.833, 200.616, 34.928, -118.915, -415]
  MoveL 5111 to (-60.1, -32.82, -121.08) mm, rotated rx -9.61 ry -16.54 rz -54.03 deg; joints [-9.844, -64.294, 113.974, 200.607, 34.941, -118.906, -415]
  MoveL 5112 to (-58.98, -34.54, -121.03) mm, rotated rx -9.61 ry -16.54 rz -54.03 deg; joints [-9.849, -64.428, 114.123, 200.592, 34.953, -118.892, -415]
  MoveL 5113 to (-57.82, -36.33, -121.01) mm, rotated rx -9.61 ry -16.54 rz -54.03 deg; joints [-9.856, -64.567, 114.277, 200.573, 34.965, -118.876, -415]
  MoveL 5114 to (-56.66, -38.11, -120.89) mm, rotated rx -9.61 ry -16.54 rz -54.03 deg; joints [-9.858, -64.706, 114.43, 200.562, 34.978, -118.864, -415]
  MoveL 5115 to (-55.42, -40.03, -120.63) mm, rotated rx -9.61 ry -16.54 rz -54.03 deg; joints [-9.856, -64.857, 114.596, 200.559, 34.992, -118.858, -415]
  MoveL 5116 to (-54.1, -42.04, -120.45) mm, rotated rx -9.61 ry -16.54 rz -54.03 deg; joints [-9.856, -65.015, 114.769, 200.55, 35.007, -118.847, -415]
  MoveL 5117 to (-52.82, -43.99, -120.25) mm, rotated rx -9.61 ry -16.54 rz -54.03 deg; joints [-9.856, -65.168, 114.938, 200.543, 35.022, -118.838, -415]
  MoveL 5118 to (-51.65, -45.77, -120.13) mm, rotated rx -9.61 ry -16.54 rz -54.03 deg; joints [-9.859, -65.308, 115.092, 200.531, 35.034, -118.827, -415]
  MoveL 5119 to (-49.32, -49.29, -119.86) mm, rotated rx -9.61 ry -16.54 rz -54.03 deg; joints [-9.862, -65.585, 115.396, 200.512, 35.058, -118.807, -415]
  MoveL 5120 to (-48.13, -51.11, -119.79) mm, rotated rx -9.61 ry -16.54 rz -54.03 deg; joints [-9.867, -65.728, 115.551, 200.498, 35.068, -118.794, -415]
  MoveL 5121 to (-46.94, -52.88, -119.57) mm, rotated rx -9.61 ry -16.54 rz -54.03 deg; joints [-9.866, -65.868, 115.705, 200.494, 35.082, -118.787, -415]
  MoveL 5122 to (-45.76, -54.63, -119.41) mm, rotated rx -9.61 ry -16.54 rz -54.03 deg; joints [-9.866, -66.007, 115.857, 200.486, 35.094, -118.778, -415]
  MoveL 5123 to (-44.58, -56.38, -119.23) mm, rotated rx -9.61 ry -16.54 rz -54.03 deg; joints [-9.866, -66.146, 116.009, 200.479, 35.107, -118.77, -415]
  MoveL 5124 to (-43.37, -58.2, -119.14) mm, rotated rx -9.61 ry -16.54 rz -54.03 deg; joints [-9.87, -66.289, 116.164, 200.467, 35.117, -118.759, -415]
  MoveL 5125 to (-42.1, -60.08, -119.01) mm, rotated rx -9.61 ry -16.54 rz -54.03 deg; joints [-9.873, -66.438, 116.327, 200.456, 35.13, -118.748, -415]
  MoveL 5126 to (-41.06, -61.67, -118.95) mm, rotated rx -9.61 ry -16.54 rz -54.03 deg; joints [-9.877, -66.564, 116.461, 200.445, 35.136, -118.738, -415]
  MoveL 5127 to (-40.5, -61.31, -118.06) mm, rotated rx -9.61 ry -16.54 rz -54.03 deg; joints [-9.84, -66.551, 116.499, 200.479, 35.192, -118.746, -415]
  MoveL 5128 to (-40.48, -60.95, -117.65) mm, rotated rx -9.61 ry -16.54 rz -54.03 deg; joints [-9.822, -66.529, 116.492, 200.502, 35.21, -118.756, -415]
  MoveL 5129 to (-40.44, -60.9, -117.37) mm, rotated rx -9.61 ry -16.54 rz -54.03 deg; joints [-9.81, -66.527, 116.496, 200.518, 35.218, -118.765, -415]
  MoveL 5130 to (-40.39, -61.22, -117.26) mm, rotated rx -9.61 ry -16.54 rz -54.03 deg; joints [-9.806, -66.551, 116.511, 200.529, 35.212, -118.774, -415]
  MoveL 5131 to (-40.36, -61.67, -117.19) mm, rotated rx -9.61 ry -16.54 rz -54.03 deg; joints [-9.804, -66.582, 116.529, 200.538, 35.199, -118.785, -415]
  MoveL 5132 to (-40.34, -62.23, -117.16) mm, rotated rx -9.61 ry -16.54 rz -54.03 deg; joints [-9.804, -66.621, 116.549, 200.548, 35.182, -118.796, -415]
  MoveL 5133 to (-40.33, -62.93, -117.12) mm, rotated rx -9.61 ry -16.54 rz -54.03 deg; joints [-9.804, -66.669, 116.574, 200.56, 35.16, -118.811, -415]
  MoveL 5134 to (-40.32, -63.56, -117.1) mm, rotated rx -9.61 ry -16.54 rz -54.03 deg; joints [-9.804, -66.712, 116.595, 200.571, 35.139, -118.824, -415]
  MoveL 5135 to (-40.33, -64.08, -117.1) mm, rotated rx -9.61 ry -16.54 rz -54.03 deg; joints [-9.805, -66.748, 116.612, 200.579, 35.121, -118.835, -415]
  MoveL 5136 to (-40.32, -64.57, -117.08) mm, rotated rx -9.61 ry -16.54 rz -54.03 deg; joints [-9.805, -66.782, 116.628, 200.587, 35.105, -118.845, -415]
  MoveL 5137 to (-40.28, -65.61, -117) mm, rotated rx -9.61 ry -16.54 rz -54.03 deg; joints [-9.804, -66.854, 116.666, 200.606, 35.073, -118.867, -415]
  MoveL 5138 to (-40.25, -66.17, -116.95) mm, rotated rx -9.61 ry -16.54 rz -54.03 deg; joints [-9.803, -66.893, 116.687, 200.616, 35.056, -118.879, -415]
  MoveL 5139 to (-40.21, -66.68, -116.89) mm, rotated rx -9.61 ry -16.54 rz -54.03 deg; joints [-9.802, -66.928, 116.707, 200.627, 35.042, -118.89, -415]
  MoveL 5140 to (-40.17, -67.14, -116.81) mm, rotated rx -9.61 ry -16.54 rz -54.03 deg; joints [-9.8, -66.961, 116.726, 200.637, 35.03, -118.901, -415]
  MoveL 5141 to (-40.14, -67.6, -116.75) mm, rotated rx -9.61 ry -16.54 rz -54.03 deg; joints [-9.798, -66.994, 116.744, 200.647, 35.016, -118.911, -415]
  MoveL 5142 to (-40.12, -68.09, -116.72) mm, rotated rx -9.61 ry -16.54 rz -54.03 deg; joints [-9.798, -67.027, 116.761, 200.655, 35.001, -118.922, -415]
  MoveL 5143 to (-40.11, -68.61, -116.7) mm, rotated rx -9.61 ry -16.54 rz -54.03 deg; joints [-9.798, -67.063, 116.779, 200.664, 34.984, -118.933, -415]
  MoveL 5144 to (-40.15, -72.28, -116.7) mm, rotated rx -9.61 ry -16.54 rz -54.03 deg; joints [-9.805, -67.313, 116.893, 200.721, 34.856, -119.009, -415]
  MoveL 5145 to (-40.28, -73.9, -116.72) mm, rotated rx -9.61 ry -16.54 rz -54.03 deg; joints [-9.809, -67.422, 116.935, 200.749, 34.792, -119.046, -415]
  MoveL 5146 to (-40.42, -74.46, -116.75) mm, rotated rx -9.61 ry -16.54 rz -54.03 deg; joints [-9.811, -67.458, 116.942, 200.761, 34.765, -119.062, -415]
  MoveL 5147 to (-40.6, -74.86, -116.78) mm, rotated rx -9.61 ry -16.54 rz -54.03 deg; joints [-9.813, -67.482, 116.941, 200.771, 34.74, -119.076, -415]
  MoveL 5148 to (-40.81, -75.13, -116.83) mm, rotated rx -9.61 ry -16.54 rz -54.03 deg; joints [-9.814, -67.497, 116.932, 200.78, 34.718, -119.089, -415]
  MoveL 5149 to (-40.93, -75.21, -116.85) mm, rotated rx -9.61 ry -16.54 rz -54.03 deg; joints [-9.815, -67.5, 116.925, 200.784, 34.708, -119.095, -415]
  MoveL 5150 to (-41.06, -75.26, -116.87) mm, rotated rx -9.61 ry -16.54 rz -54.03 deg; joints [-9.816, -67.502, 116.916, 200.788, 34.698, -119.1, -415]
  MoveL 5151 to (-41.2, -75.28, -116.9) mm, rotated rx -9.61 ry -16.54 rz -54.03 deg; joints [-9.816, -67.501, 116.906, 200.792, 34.69, -119.105, -415]
  MoveL 5152 to (-41.34, -75.28, -116.93) mm, rotated rx -9.61 ry -16.54 rz -54.03 deg; joints [-9.817, -67.498, 116.895, 200.795, 34.681, -119.11, -415]
  MoveL 5153 to (-41.65, -75.19, -116.99) mm, rotated rx -9.61 ry -16.54 rz -54.03 deg; joints [-9.819, -67.487, 116.868, 200.801, 34.666, -119.118, -415]
  MoveL 5154 to (-42.31, -74.76, -117.12) mm, rotated rx -9.61 ry -16.54 rz -54.03 deg; joints [-9.821, -67.445, 116.801, 200.81, 34.642, -119.132, -415]
  MoveL 5155 to (-43.02, -74.05, -117.26) mm, rotated rx -9.61 ry -16.54 rz -54.03 deg; joints [-9.823, -67.385, 116.721, 200.816, 34.624, -119.141, -415]
  MoveL 5156 to (-44.45, -72.19, -117.53) mm, rotated rx -9.61 ry -16.54 rz -54.03 deg; joints [-9.826, -67.233, 116.548, 200.823, 34.603, -119.152, -415]
  MoveL 5157 to (-45.79, -70.18, -117.77) mm, rotated rx -9.61 ry -16.54 rz -54.03 deg; joints [-9.828, -67.073, 116.377, 200.826, 34.592, -119.157, -415]
  MoveL 5158 to (-75.46, -25.08, -122.85) mm, rotated rx -9.61 ry -16.54 rz -54.03 deg; joints [-9.851, -63.517, 112.474, 200.968, 34.262, -119.351, -415]
  MoveL 5159 to (-77.56, -21.88, -123.22) mm, rotated rx -9.61 ry -16.54 rz -54.03 deg; joints [-9.853, -63.267, 112.19, 200.983, 34.231, -119.37, -415]
  MoveL 5160 to (-79.47, -18.65, -123.63) mm, rotated rx -9.61 ry -16.54 rz -54.03 deg; joints [-9.857, -63.018, 111.92, 200.986, 34.21, -119.379, -415]
  MoveL 5161 to (-79.98, -17.25, -123.84) mm, rotated rx -9.61 ry -16.54 rz -54.03 deg; joints [-9.861, -62.915, 111.827, 200.974, 34.218, -119.367, -415]
  MoveL 5162 to (-80.02, -16.7, -123.94) mm, rotated rx -9.61 ry -16.54 rz -54.03 deg; joints [-9.864, -62.877, 111.804, 200.962, 34.231, -119.356, -415]
  MoveL 5163 to (-79.97, -16.48, -123.98) mm, rotated rx -9.61 ry -16.54 rz -54.03 deg; joints [-9.866, -62.863, 111.799, 200.954, 34.24, -119.348, -415]
  MoveL 5164 to (-79.87, -16.3, -124.02) mm, rotated rx -9.61 ry -16.54 rz -54.03 deg; joints [-9.867, -62.852, 111.8, 200.945, 34.25, -119.338, -415]
  MoveL 5165 to (-79.71, -16.16, -124.06) mm, rotated rx -9.61 ry -16.54 rz -54.03 deg; joints [-9.869, -62.845, 111.807, 200.935, 34.263, -119.328, -415]
  MoveL 5166 to (-79.5, -16.06, -124.09) mm, rotated rx -9.61 ry -16.54 rz -54.03 deg; joints [-9.871, -62.842, 111.82, 200.924, 34.277, -119.315, -415]
  MoveL 5167 to (-79.23, -16.02, -124.12) mm, rotated rx -9.61 ry -16.54 rz -54.03 deg; joints [-9.873, -62.844, 111.84, 200.91, 34.294, -119.301, -415]
  MoveL 5168 to (-78.89, -16.03, -124.15) mm, rotated rx -9.61 ry -16.54 rz -54.03 deg; joints [-9.875, -62.85, 111.868, 200.896, 34.314, -119.285, -415]
  MoveL 5169 to (-76.79, -16.66, -124.2) mm, rotated rx -9.61 ry -16.54 rz -54.03 deg; joints [-9.886, -62.926, 112.057, 200.82, 34.417, -119.203, -415]
  MoveL 5170 to (-74.86, -17.48, -124.2) mm, rotated rx -9.61 ry -16.54 rz -54.03 deg; joints [-9.894, -63.013, 112.24, 200.757, 34.505, -119.134, -415]
  MoveL 5171 to (-71.56, -19.38, -124.24) mm, rotated rx -9.61 ry -16.54 rz -54.03 deg; joints [-9.91, -63.193, 112.569, 200.653, 34.64, -119.023, -415]
  MoveL 5172 to (-68.95, -21.77, -124.35) mm, rotated rx -9.61 ry -16.54 rz -54.03 deg; joints [-9.929, -63.395, 112.86, 200.578, 34.72, -118.949, -415]
  MoveL 5173 to (-65.63, -26.83, -124.65) mm, rotated rx -9.61 ry -16.54 rz -54.03 deg; joints [-9.963, -63.786, 113.3, 200.498, 34.757, -118.883, -415]
  MoveL 5174 to (-64.77, -29.03, -124.78) mm, rotated rx -9.61 ry -16.54 rz -54.03 deg; joints [-9.975, -63.947, 113.444, 200.485, 34.738, -118.879, -415]
  MoveL 5175 to (-53.51, -61.93, -126.65) mm, rotated rx -9.61 ry -16.54 rz -54.03 deg; joints [-10.163, -66.343, 115.431, 200.383, 34.313, -118.928, -415]
  MoveL 5176 to (-52.54, -64.74, -126.81) mm, rotated rx -9.61 ry -16.54 rz -54.03 deg; joints [-10.18, -66.549, 115.598, 200.376, 34.273, -118.934, -415]
  MoveL 5177 to (-50.89, -68.09, -127.05) mm, rotated rx -9.61 ry -16.54 rz -54.03 deg; joints [-10.203, -66.802, 115.834, 200.345, 34.251, -118.919, -415]
  MoveL 5178 to (-49.96, -69.24, -127.19) mm, rotated rx -9.61 ry -16.54 rz -54.03 deg; joints [-10.215, -66.895, 115.943, 200.317, 34.263, -118.896, -415]
  MoveL 5179 to (-49.5, -69.55, -127.26) mm, rotated rx -9.61 ry -16.54 rz -54.03 deg; joints [-10.221, -66.923, 115.988, 200.3, 34.278, -118.88, -415]
  MoveL 5180 to (-49.29, -69.61, -127.3) mm, rotated rx -9.61 ry -16.54 rz -54.03 deg; joints [-10.223, -66.931, 116.007, 200.29, 34.288, -118.87, -415]
  MoveL 5181 to (-49.08, -69.62, -127.33) mm, rotated rx -9.61 ry -16.54 rz -54.03 deg; joints [-10.226, -66.935, 116.023, 200.28, 34.299, -118.86, -415]
  MoveL 5182 to (-48.88, -69.55, -127.37) mm, rotated rx -9.61 ry -16.54 rz -54.03 deg; joints [-10.228, -66.934, 116.036, 200.269, 34.312, -118.849, -415]
  MoveL 5183 to (-48.69, -69.41, -127.4) mm, rotated rx -9.61 ry -16.54 rz -54.03 deg; joints [-10.229, -66.927, 116.046, 200.258, 34.327, -118.837, -415]
  MoveL 5184 to (-48.51, -69.19, -127.44) mm, rotated rx -9.61 ry -16.54 rz -54.03 deg; joints [-10.231, -66.915, 116.053, 200.246, 34.344, -118.824, -415]
  MoveL 5185 to (-48.35, -68.89, -127.47) mm, rotated rx -9.61 ry -16.54 rz -54.03 deg; joints [-10.232, -66.897, 116.056, 200.233, 34.364, -118.809, -415]
  MoveL 5186 to (-47.87, -66.75, -127.59) mm, rotated rx -9.61 ry -16.54 rz -54.03 deg; joints [-10.235, -66.759, 116.023, 200.176, 34.462, -118.742, -415]
  MoveL 5187 to (-47.81, -66.24, -127.61) mm, rotated rx -9.61 ry -16.54 rz -54.03 deg; joints [-10.235, -66.725, 116.011, 200.165, 34.483, -118.729, -415]
  MoveL 5188 to (-47.79, -65.78, -127.66) mm, rotated rx -9.61 ry -16.54 rz -54.03 deg; joints [-10.236, -66.694, 115.998, 200.154, 34.499, -118.717, -415]
  MoveL 5189 to (-47.78, -65.34, -127.73) mm, rotated rx -9.61 ry -16.54 rz -54.03 deg; joints [-10.238, -66.663, 115.983, 200.143, 34.513, -118.705, -415]
  MoveL 5190 to (-47.76, -64.89, -127.79) mm, rotated rx -9.61 ry -16.54 rz -54.03 deg; joints [-10.239, -66.633, 115.97, 200.132, 34.529, -118.693, -415]
  MoveL 5191 to (-47.73, -64.43, -127.82) mm, rotated rx -9.61 ry -16.54 rz -54.03 deg; joints [-10.24, -66.602, 115.957, 200.122, 34.546, -118.682, -415]
  MoveL 5192 to (-47.09, -59.79, -127.83) mm, rotated rx -9.61 ry -16.54 rz -54.03 deg; joints [-10.233, -66.297, 115.855, 200.033, 34.739, -118.567, -415]
  MoveL 5193 to (-47.04, -59.35, -127.86) mm, rotated rx -9.61 ry -16.54 rz -54.03 deg; joints [-10.233, -66.268, 115.844, 200.024, 34.756, -118.556, -415]
  MoveL 5194 to (-46.98, -58.88, -127.87) mm, rotated rx -9.61 ry -16.54 rz -54.03 deg; joints [-10.232, -66.237, 115.833, 200.014, 34.775, -118.544, -415]
  MoveL 5195 to (-46.84, -57.85, -127.87) mm, rotated rx -9.61 ry -16.54 rz -54.03 deg; joints [-10.231, -66.169, 115.81, 199.995, 34.817, -118.519, -415]
  MoveL 5196 to (-46.77, -57.28, -127.88) mm, rotated rx -9.61 ry -16.54 rz -54.03 deg; joints [-10.23, -66.131, 115.797, 199.984, 34.84, -118.505, -415]
  MoveL 5197 to (-46.72, -56.68, -127.89) mm, rotated rx -9.61 ry -16.54 rz -54.03 deg; joints [-10.23, -66.091, 115.781, 199.973, 34.863, -118.491, -415]
  MoveL 5198 to (-46.7, -56.02, -127.92) mm, rotated rx -9.61 ry -16.54 rz -54.03 deg; joints [-10.229, -66.047, 115.76, 199.962, 34.885, -118.477, -415]
  MoveL 5199 to (-46.76, -55.36, -127.95) mm, rotated rx -9.61 ry -16.54 rz -54.03 deg; joints [-10.229, -66.001, 115.733, 199.953, 34.904, -118.466, -415]
  MoveL 5200 to (-46.87, -54.72, -127.96) mm, rotated rx -9.61 ry -16.54 rz -54.03 deg; joints [-10.228, -65.955, 115.703, 199.948, 34.918, -118.458, -415]
  MoveL 5201 to (-46.94, -56.03, -128.94) mm, rotated rx -9.61 ry -16.54 rz -54.03 deg; joints [-10.272, -66.038, 115.733, 199.901, 34.858, -118.443, -415]
  MoveL 5202 to (-47.8, -55, -129.37) mm, rotated rx -9.61 ry -16.54 rz -54.03 deg; joints [-10.285, -65.952, 115.628, 199.89, 34.837, -118.441, -415]
  MoveL 5203 to (-48.64, -53.77, -129.69) mm, rotated rx -9.61 ry -16.54 rz -54.03 deg; joints [-10.293, -65.854, 115.518, 199.882, 34.825, -118.439, -415]
  MoveL 5204 to (-49.5, -52.31, -129.92) mm, rotated rx -9.61 ry -16.54 rz -54.03 deg; joints [-10.296, -65.74, 115.4, 199.879, 34.82, -118.438, -415]
  MoveL 5205 to (-50.48, -50.41, -130.14) mm, rotated rx -9.61 ry -16.54 rz -54.03 deg; joints [-10.297, -65.594, 115.258, 199.875, 34.823, -118.435, -415]
  MoveL 5206 to (-51.43, -48.5, -130.25) mm, rotated rx -9.61 ry -16.54 rz -54.03 deg; joints [-10.295, -65.449, 115.118, 199.877, 34.829, -118.435, -415]
  MoveL 5207 to (-52.38, -46.59, -130.36) mm, rotated rx -9.61 ry -16.54 rz -54.03 deg; joints [-10.291, -65.304, 114.977, 199.88, 34.834, -118.435, -415]
  MoveL 5208 to (-53.35, -44.68, -130.59) mm, rotated rx -9.61 ry -16.54 rz -54.03 deg; joints [-10.293, -65.158, 114.835, 199.875, 34.837, -118.431, -415]
  MoveL 5209 to (-54.29, -42.77, -130.71) mm, rotated rx -9.61 ry -16.54 rz -54.03 deg; joints [-10.291, -65.013, 114.695, 199.877, 34.842, -118.431, -415]
  MoveL 5210 to (-55.24, -40.86, -130.94) mm, rotated rx -9.61 ry -16.54 rz -54.03 deg; joints [-10.293, -64.868, 114.553, 199.872, 34.844, -118.427, -415]
  MoveL 5211 to (-56.18, -38.95, -131.06) mm, rotated rx -9.61 ry -16.54 rz -54.03 deg; joints [-10.29, -64.723, 114.412, 199.874, 34.849, -118.427, -415]
  MoveL 5212 to (-57.12, -37.03, -131.18) mm, rotated rx -9.61 ry -16.54 rz -54.03 deg; joints [-10.287, -64.578, 114.271, 199.877, 34.853, -118.428, -415]
  MoveL 5213 to (-58.06, -35.11, -131.41) mm, rotated rx -9.61 ry -16.54 rz -54.03 deg; joints [-10.29, -64.432, 114.129, 199.871, 34.856, -118.423, -415]
  MoveL 5214 to (-58.94, -33.27, -131.52) mm, rotated rx -9.61 ry -16.54 rz -54.03 deg; joints [-10.287, -64.294, 113.995, 199.874, 34.861, -118.424, -415]
  MoveL 5215 to (-59.79, -31.48, -131.72) mm, rotated rx -9.61 ry -16.54 rz -54.03 deg; joints [-10.288, -64.158, 113.863, 199.87, 34.864, -118.42, -415]
  MoveL 5216 to (-60.84, -29.35, -131.88) mm, rotated rx -9.61 ry -16.54 rz -54.03 deg; joints [-10.287, -63.998, 113.705, 199.871, 34.867, -118.42, -415]
  MoveL 5217 to (-62, -26.89, -131.97) mm, rotated rx -9.61 ry -16.54 rz -54.03 deg; joints [-10.281, -63.813, 113.526, 199.878, 34.873, -118.423, -415]
  MoveL 5218 to (-62.9, -25.02, -132.04) mm, rotated rx -9.61 ry -16.54 rz -54.03 deg; joints [-10.276, -63.673, 113.388, 199.884, 34.877, -118.426, -415]
  MoveL 5219 to (-63.74, -23.28, -132.17) mm, rotated rx -9.61 ry -16.54 rz -54.03 deg; joints [-10.275, -63.542, 113.259, 199.886, 34.879, -118.427, -415]
  MoveL 5220 to (-64.6, -21.5, -132.27) mm, rotated rx -9.61 ry -16.54 rz -54.03 deg; joints [-10.272, -63.408, 113.127, 199.889, 34.881, -118.429, -415]
  MoveL 5221 to (-65.44, -19.73, -132.38) mm, rotated rx -9.61 ry -16.54 rz -54.03 deg; joints [-10.27, -63.276, 112.997, 199.892, 34.883, -118.43, -415]
  MoveL 5222 to (-66.33, -17.88, -132.45) mm, rotated rx -9.61 ry -16.54 rz -54.03 deg; joints [-10.266, -63.137, 112.859, 199.898, 34.886, -118.433, -415]
  MoveL 5223 to (-67.28, -15.87, -132.55) mm, rotated rx -9.61 ry -16.54 rz -54.03 deg; joints [-10.262, -62.987, 112.711, 199.903, 34.888, -118.436, -415]
  MoveL 5224 to (-68.29, -13.68, -132.81) mm, rotated rx -9.61 ry -16.54 rz -54.03 deg; joints [-10.265, -62.823, 112.55, 199.898, 34.89, -118.432, -415]
  MoveL 5225 to (-69.67, -11.92, -133.8) mm, rotated rx -9.61 ry -16.54 rz -54.03 deg; joints [-10.296, -62.678, 112.368, 199.864, 34.848, -118.42, -415]
  MoveL 5226 to (-68.7, -12.51, -134.28) mm, rotated rx -9.61 ry -16.54 rz -54.03 deg; joints [-10.321, -62.731, 112.462, 199.803, 34.882, -118.369, -415]
  MoveL 5227 to (-68.18, -12.81, -134.59) mm, rotated rx -9.61 ry -16.54 rz -54.03 deg; joints [-10.337, -62.758, 112.511, 199.767, 34.9, -118.339, -415]
  MoveL 5228 to (-68.09, -12.86, -134.74) mm, rotated rx -9.61 ry -16.54 rz -54.03 deg; joints [-10.343, -62.761, 112.518, 199.754, 34.901, -118.33, -415]
  MoveL 5229 to (-68.39, -12.68, -134.78) mm, rotated rx -9.61 ry -16.54 rz -54.03 deg; joints [-10.343, -62.744, 112.488, 199.761, 34.889, -118.338, -415]
  MoveL 5230 to (-68.79, -12.44, -134.8) mm, rotated rx -9.61 ry -16.54 rz -54.03 deg; joints [-10.342, -62.722, 112.448, 199.772, 34.872, -118.35, -415]
  MoveL 5231 to (-69.19, -12.18, -134.83) mm, rotated rx -9.61 ry -16.54 rz -54.03 deg; joints [-10.341, -62.698, 112.406, 199.781, 34.856, -118.361, -415]
  MoveL 5232 to (-69.56, -11.92, -134.89) mm, rotated rx -9.61 ry -16.54 rz -54.03 deg; joints [-10.342, -62.675, 112.367, 199.788, 34.841, -118.37, -415]
  MoveL 5233 to (-69.95, -11.67, -134.93) mm, rotated rx -9.61 ry -16.54 rz -54.03 deg; joints [-10.342, -62.651, 112.327, 199.796, 34.825, -118.38, -415]
  MoveL 5234 to (-70.37, -11.41, -134.95) mm, rotated rx -9.61 ry -16.54 rz -54.03 deg; joints [-10.34, -62.627, 112.285, 199.808, 34.808, -118.393, -415]
  MoveL 5235 to (-72.63, -10.09, -134.95) mm, rotated rx -9.61 ry -16.54 rz -54.03 deg; joints [-10.329, -62.503, 112.057, 199.876, 34.713, -118.466, -415]
  MoveL 5236 to (-73.02, -9.85, -134.97) mm, rotated rx -9.61 ry -16.54 rz -54.03 deg; joints [-10.328, -62.481, 112.018, 199.886, 34.697, -118.477, -415]
  MoveL 5237 to (-73.34, -9.63, -135.01) mm, rotated rx -9.61 ry -16.54 rz -54.03 deg; joints [-10.328, -62.461, 111.984, 199.894, 34.684, -118.486, -415]
  MoveL 5238 to (-73.73, -9.39, -135.03) mm, rotated rx -9.61 ry -16.54 rz -54.03 deg; joints [-10.327, -62.439, 111.944, 199.904, 34.668, -118.497, -415]
  MoveL 5239 to (-74.24, -9.07, -135.05) mm, rotated rx -9.61 ry -16.54 rz -54.03 deg; joints [-10.325, -62.409, 111.892, 199.918, 34.647, -118.513, -415]
  MoveL 5240 to (-74.84, -8.67, -135.1) mm, rotated rx -9.61 ry -16.54 rz -54.03 deg; joints [-10.325, -62.373, 111.829, 199.932, 34.622, -118.529, -415]
  MoveL 5241 to (-75.36, -8.35, -135.13) mm, rotated rx -9.61 ry -16.54 rz -54.03 deg; joints [-10.323, -62.343, 111.775, 199.946, 34.601, -118.545, -415]
  MoveL 5242 to (-75.82, -8.08, -135.13) mm, rotated rx -9.61 ry -16.54 rz -54.03 deg; joints [-10.321, -62.317, 111.729, 199.96, 34.581, -118.56, -415]
  MoveL 5243 to (-77.18, -7.28, -135.13) mm, rotated rx -9.61 ry -16.54 rz -54.03 deg; joints [-10.315, -62.243, 111.592, 200.001, 34.524, -118.604, -415]
  MoveL 5244 to (-79.54, -5.57, -135.48) mm, rotated rx -9.61 ry -16.54 rz -54.03 deg; joints [-10.316, -62.089, 111.339, 200.048, 34.431, -118.662, -415]
  MoveL 5245 to (-80.42, -4.62, -135.9) mm, rotated rx -9.61 ry -16.54 rz -54.03 deg; joints [-10.329, -62.009, 111.23, 200.042, 34.4, -118.667, -415]
  MoveL 5246 to (-81.12, -3.62, -136.5) mm, rotated rx -9.61 ry -16.54 rz -54.03 deg; joints [-10.349, -61.928, 111.132, 200.018, 34.38, -118.656, -415]
  MoveL 5247 to (-81.93, -1.45, -138.21) mm, rotated rx -9.61 ry -16.54 rz -54.03 deg; joints [-10.411, -61.762, 110.972, 199.912, 34.372, -118.584, -415]
  MoveL 5248 to (-81.96, 0.96, -140.61) mm, rotated rx -9.61 ry -16.54 rz -54.03 deg; joints [-10.503, -61.589, 110.858, 199.73, 34.406, -118.449, -415]
  MoveL 5249 to (-81.34, 2.92, -143) mm, rotated rx -9.61 ry -16.54 rz -54.03 deg; joints [-10.598, -61.456, 110.812, 199.53, 34.467, -118.294, -415]
  MoveL 5250 to (-80.83, 3.49, -143.95) mm, rotated rx -9.61 ry -16.54 rz -54.03 deg; joints [-10.637, -61.422, 110.823, 199.444, 34.502, -118.225, -415]
  MoveL 5251 to (-80.18, 3.77, -144.72) mm, rotated rx -9.61 ry -16.54 rz -54.03 deg; joints [-10.67, -61.409, 110.857, 199.367, 34.538, -118.162, -415]
  MoveL 5252 to (-79.8, 3.81, -145.04) mm, rotated rx -9.61 ry -16.54 rz -54.03 deg; joints [-10.685, -61.411, 110.882, 199.332, 34.557, -118.132, -415]
  MoveL 5253 to (-79.39, 3.78, -145.31) mm, rotated rx -9.61 ry -16.54 rz -54.03 deg; joints [-10.698, -61.418, 110.913, 199.299, 34.577, -118.104, -415]
  MoveL 5254 to (-78.47, 3.51, -145.74) mm, rotated rx -9.61 ry -16.54 rz -54.03 deg; joints [-10.719, -61.449, 110.992, 199.24, 34.619, -118.053, -415]
  MoveL 5255 to (-77.42, 2.96, -146) mm, rotated rx -9.61 ry -16.54 rz -54.03 deg; joints [-10.735, -61.501, 111.094, 199.19, 34.662, -118.007, -415]
  MoveL 5256 to (-76.23, 2.13, -146.08) mm, rotated rx -9.61 ry -16.54 rz -54.03 deg; joints [-10.745, -61.574, 111.219, 199.15, 34.709, -117.967, -415]
  MoveL 5257 to (-75.81, 1.81, -146.08) mm, rotated rx -9.61 ry -16.54 rz -54.03 deg; joints [-10.747, -61.602, 111.263, 199.138, 34.724, -117.955, -415]
